LIN {X -0.046,Y -193.503,Z 910.176,A 0.000,B 0.000,C 90.000,E1 31.671} C_DIS
LIN {X 0.056,Y -188.124,Z 910.158,A 0.000,B 0.000,C 90.000,E1 28.359} C_DIS
LIN {X 0.087,Y -183.389,Z 910.139,A 0.000,B 0.000,C 90.000,E1 25.027} C_DIS
LIN {X -0.058,Y -179.252,Z 910.121,A 0.000,B 0.000,C 90.000,E1 21.716} C_DIS
LIN {X 0.005,Y -175.085,Z 910.097,A 0.000,B 0.000,C 90.000,E1 17.457} C_DIS
LIN {X 0.015,Y -172.098,Z 910.073,A 0.000,B 0.000,C 90.000,E1 13.175} C_DIS
LIN {X 0.060,Y -169.577,Z 910.040,A 0.000,B 0.000,C 90.000,E1 7.125} C_DIS
LIN {X 0.074,Y -170.579,Z 909.973,A 0.000,B 0.000,C 90.000,E1 355.179} C_DIS
LIN {X -0.024,Y -173.354,Z 909.945,A 0.000,B 0.000,C 90.000,E1 350.038} C_DIS
LIN {X -0.023,Y -176.708,Z 909.921,A 0.000,B 0.000,C 90.000,E1 345.755} C_DIS
LIN {X -0.051,Y -180.143,Z 909.902,A 0.000,B 0.000,C 90.000,E1 342.362} C_DIS
LIN {X 0.058,Y -184.300,Z 909.883,A 0.000,B 0.000,C 90.000,E1 338.954} C_DIS
LIN {X 0.061,Y -189.349,Z 909.865,A 0.000,B 0.000,C 90.000,E1 335.613} C_DIS
LIN {X -0.101,Y -195.206,Z 909.846,A 0.000,B 0.000,C 90.000,E1 332.359} C_DIS
LIN {X 0.047,Y -203.252,Z 909.824,A 0.000,B 0.000,C 90.000,E1 328.250} C_DIS
LIN {X 0.026,Y -210.215,Z 909.806,A 0.000,B 0.000,C 90.000,E1 325.055} C_DIS
LIN {X 0.020,Y -217.690,Z 909.788,A 0.000,B 0.000,C 90.000,E1 321.904} C_DIS
LIN {X 0.091,Y -226.821,Z 909.769,A 0.000,B 0.000,C 90.000,E1 318.405} C_DIS
LIN {X -0.057,Y -235.880,Z 909.752,A 0.000,B 0.000,C 90.000,E1 315.405} C_DIS
LIN {X 0.035,Y -245.907,Z 909.736,A 0.000,B 0.000,C 90.000,E1 312.405} C_DIS
LIN {X 0.057,Y -257.101,Z 909.719,A 0.000,B 0.000,C 90.000,E1 309.483} C_DIS
LIN {X -0.096,Y -269.400,Z 909.704,A 0.000,B 0.000,C 90.000,E1 306.664} C_DIS
LIN {X 0.083,Y -284.961,Z 909.686,A 0.000,B 0.000,C 90.000,E1 303.499} C_DIS
LIN {X 0.101,Y -301.959,Z 909.669,A 0.000,B 0.000,C 90.000,E1 300.463} C_DIS
LIN {X 0.029,Y -316.328,Z 909.657,A 0.000,B 0.000,C 90.000,E1 298.180} C_DIS
LIN {X -0.108,Y -329.854,Z 909.646,A 0.000,B 0.000,C 90.000,E1 296.283} C_DIS
LIN {X 0.009,Y -344.391,Z 909.635,A 0.000,B 0.000,C 90.000,E1 294.387} C_DIS
LIN {X 0.127,Y -367.738,Z 909.620,A 0.000,B 0.000,C 90.000,E1 291.663} C_DIS
LIN {X -0.013,Y -383.531,Z 909.611,A 0.000,B 0.000,C 90.000,E1 289.993} C_DIS
LIN {X -0.045,Y -401.556,Z 909.601,A 0.000,B 0.000,C 90.000,E1 288.109} C_DIS
LIN {X 0.162,Y -414.278,Z 909.593,A 0.000,B 0.000,C 90.000,E1 286.732} C_DIS
LIN {X 0.078,Y -424.276,Z 909.587,A 0.000,B 0.000,C 90.000,E1 285.662} C_DIS
LIN {X 0.006,Y -433.925,Z 909.581,A 0.000,B 0.000,C 90.000,E1 284.592} C_DIS
LIN {X 0.143,Y -445.299,Z 909.574,A 0.000,B 0.000,C 90.000,E1 283.244} C_DIS
LIN {X -0.231,Y -453.814,Z 909.568,A 0.000,B 0.000,C 90.000,E1 282.243} C_DIS
LIN {X -0.069,Y -461.769,Z 909.562,A 0.000,B 0.000,C 90.000,E1 281.186} C_DIS
LIN {X -0.046,Y -471.069,Z 909.555,A 0.000,B 0.000,C 90.000,E1 279.905} C_DIS
LIN {X -0.097,Y -476.327,Z 909.551,A 0.000,B 0.000,C 90.000,E1 279.151} C_DIS
LIN {X -0.096,Y -480.913,Z 909.547,A 0.000,B 0.000,C 90.000,E1 278.398} C_DIS
LIN {X -0.059,Y -484.725,Z 909.542,A 0.000,B 0.000,C 90.000,E1 277.644} C_DIS
LIN {X 0.126,Y -486.841,Z 909.540,A 0.000,B 0.000,C 90.000,E1 277.125} C_DIS
LIN {X -0.159,Y -488.603,Z 909.537,A 0.000,B 0.000,C 90.000,E1 276.663} C_DIS
LIN {X 0.047,Y -490.002,Z 909.534,A 0.000,B 0.000,C 90.000,E1 276.144} C_DIS
LIN {X -0.225,Y -491.072,Z 909.531,A 0.000,B 0.000,C 90.000,E1 275.682} C_DIS
LIN {X -0.002,Y -491.799,Z 909.529,A 0.000,B 0.000,C 90.000,E1 275.163} C_DIS
LIN {X 0.226,Y -492.165,Z 909.526,A 0.000,B 0.000,C 90.000,E1 274.645} C_DIS
LIN {X -0.070,Y -492.073,Z 909.523,A 0.000,B 0.000,C 90.000,E1 274.188} C_DIS
LIN {X 0.163,Y -491.518,Z 909.521,A 0.000,B 0.000,C 90.000,E1 273.669} C_DIS
LIN {X -0.127,Y -490.551,Z 909.518,A 0.000,B 0.000,C 90.000,E1 273.212} C_DIS
LIN {X 0.098,Y -489.016,Z 909.515,A 0.000,B 0.000,C 90.000,E1 272.694} C_DIS
LIN {X -0.195,Y -486.904,Z 909.512,A 0.000,B 0.000,C 90.000,E1 272.236} C_DIS
LIN {X 0.008,Y -484.104,Z 909.510,A 0.000,B 0.000,C 90.000,E1 271.718} C_DIS
LIN {X 0.173,Y -480.512,Z 909.507,A 0.000,B 0.000,C 90.000,E1 271.203} C_DIS
LIN {X -0.158,Y -476.050,Z 909.504,A 0.000,B 0.000,C 90.000,E1 270.745} C_DIS
LIN {X -0.032,Y -470.550,Z 909.501,A 0.000,B 0.000,C 90.000,E1 270.229} C_DIS
LIN {X -0.022,Y -464.477,Z 909.499,A 0.000,B 0.000,C 90.000,E1 269.771} C_DIS
LIN {X 0.008,Y -458.177,Z 909.497,A 0.000,B 0.000,C 90.000,E1 269.370} C_DIS
LIN {X -0.030,Y -451.593,Z 909.495,A 0.000,B 0.000,C 90.000,E1 269.026} C_DIS
LIN {X -0.148,Y -444.694,Z 909.493,A 0.000,B 0.000,C 90.000,E1 268.740} C_DIS
LIN {X 0.111,Y -437.786,Z 909.492,A 0.000,B 0.000,C 90.000,E1 268.453} C_DIS
LIN {X -0.214,Y -430.109,Z 909.490,A 0.000,B 0.000,C 90.000,E1 268.282} C_DIS
LIN {X -0.153,Y -421.664,Z 909.489,A 0.000,B 0.000,C 90.000,E1 268.108} C_DIS
LIN {X -0.161,Y -411.053,Z 909.489,A 0.000,B 0.000,C 90.000,E1 267.993} C_DIS
LIN {X 0.050,Y -404.242,Z 909.489,A 0.000,B 0.000,C 90.000,E1 267.936} C_DIS
LIN {X -0.007,Y -181.114,Z 909.489,A 0.000,B 0.000,C 90.000,E1 267.936} C_DIS
LIN {X 0.043,Y -180.906,Z 909.474,A 0.000,B 0.000,C 90.000,E1 265.355} C_DIS
LIN {X -0.063,Y -180.689,Z 909.470,A 0.000,B 0.000,C 90.000,E1 264.546} C_DIS
LIN {X 0.015,Y -178.773,Z 909.441,A 0.000,B 0.000,C 90.000,E1 259.454} C_DIS
LIN {X -0.082,Y -175.819,Z 909.413,A 0.000,B 0.000,C 90.000,E1 254.393} C_DIS
LIN {X 0.080,Y -172.006,Z 909.385,A 0.000,B 0.000,C 90.000,E1 249.209} C_DIS
LIN {X 0.055,Y -171.424,Z 909.380,A 0.000,B 0.000,C 90.000,E1 248.358} C_DIS
LIN {X -0.049,Y -167.662,Z 909.356,A 0.000,B 0.000,C 90.000,E1 244.076} C_DIS
LIN {X 0.039,Y -166.330,Z 909.346,A 0.000,B 0.000,C 90.000,E1 242.308} C_DIS
LIN {X 0.025,Y -163.069,Z 909.327,A 0.000,B 0.000,C 90.000,E1 238.820} C_DIS
LIN {X -0.064,Y -161.008,Z 909.312,A 0.000,B 0.000,C 90.000,E1 236.215} C_DIS
LIN {X 0.046,Y -157.752,Z 909.293,A 0.000,B 0.000,C 90.000,E1 232.637} C_DIS
LIN {X -0.016,Y -155.790,Z 909.278,A 0.000,B 0.000,C 90.000,E1 229.989} C_DIS
LIN {X 0.039,Y -152.044,Z 909.253,A 0.000,B 0.000,C 90.000,E1 225.486} C_DIS
LIN {X 0.057,Y -150.292,Z 909.238,A 0.000,B 0.000,C 90.000,E1 222.771} C_DIS
LIN {X -0.018,Y -147.040,Z 909.213,A 0.000,B 0.000,C 90.000,E1 218.257} C_DIS
LIN {X -0.025,Y -145.620,Z 909.197,A 0.000,B 0.000,C 90.000,E1 215.518} C_DIS
LIN {X -0.026,Y -143.004,Z 909.172,A 0.000,B 0.000,C 90.000,E1 210.924} C_DIS
LIN {X 0.031,Y -141.631,Z 909.151,A 0.000,B 0.000,C 90.000,E1 207.206} C_DIS
LIN {X -0.043,Y -139.435,Z 909.115,A 0.000,B 0.000,C 90.000,E1 200.737} C_DIS
LIN {X 0.011,Y -139.167,Z 909.105,A 0.000,B 0.000,C 90.000,E1 198.852} C_DIS
LIN {X 0.044,Y -138.316,Z 909.053,A 0.000,B 0.000,C 90.000,E1 189.500} C_DIS
LIN {X 0.055,Y -139.475,Z 909.006,A 0.000,B 0.000,C 90.000,E1 181.088} C_DIS
LIN {X -0.003,Y -141.056,Z 908.975,A 0.000,B 0.000,C 90.000,E1 175.527} C_DIS
LIN {X -0.050,Y -142.427,Z 908.960,A 0.000,B 0.000,C 90.000,E1 172.761} C_DIS
LIN {X 0.011,Y -144.665,Z 908.934,A 0.000,B 0.000,C 90.000,E1 168.117} C_DIS
LIN {X -0.005,Y -147.249,Z 908.914,A 0.000,B 0.000,C 90.000,E1 164.448} C_DIS
LIN {X 0.013,Y -150.566,Z 908.888,A 0.000,B 0.000,C 90.000,E1 159.880} C_DIS
LIN {X 0.092,Y -154.035,Z 908.868,A 0.000,B 0.000,C 90.000,E1 156.230} C_DIS
LIN {X 0.019,Y -157.451,Z 908.848,A 0.000,B 0.000,C 90.000,E1 152.666} C_DIS
LIN {X -0.032,Y -161.669,Z 908.828,A 0.000,B 0.000,C 90.000,E1 149.125} C_DIS
LIN {X -0.014,Y -165.864,Z 908.809,A 0.000,B 0.000,C 90.000,E1 145.595} C_DIS
LIN {X -0.023,Y -170.841,Z 908.789,A 0.000,B 0.000,C 90.000,E1 142.110} C_DIS
LIN {X 0.024,Y -175.711,Z 908.770,A 0.000,B 0.000,C 90.000,E1 138.647} C_DIS
LIN {X 0.015,Y -181.323,Z 908.751,A 0.000,B 0.000,C 90.000,E1 135.243} C_DIS
LIN {X -0.115,Y -186.807,Z 908.733,A 0.000,B 0.000,C 90.000,E1 131.919} C_DIS
LIN {X -0.043,Y -191.397,Z 908.719,A 0.000,B 0.000,C 90.000,E1 129.402} C_DIS
LIN {X -0.106,Y -193.630,Z 908.711,A 0.000,B 0.000,C 90.000,E1 128.096} C_DIS
LIN {X 0.018,Y -295.882,Z 908.711,A 0.000,B 0.000,C 90.000,E1 128.051} C_DIS
LIN {X 0.042,Y -297.426,Z 908.711,A 0.000,B 0.000,C 90.000,E1 128.016} C_DIS
LIN {X 0.058,Y -302.690,Z 908.710,A 0.000,B 0.000,C 90.000,E1 127.729} C_DIS
LIN {X 0.059,Y -305.900,Z 908.708,A 0.000,B 0.000,C 90.000,E1 127.397} C_DIS
LIN {X 0.025,Y -309.482,Z 908.705,A 0.000,B 0.000,C 90.000,E1 126.824} C_DIS
LIN {X -0.011,Y -310.894,Z 908.703,A 0.000,B 0.000,C 90.000,E1 126.503} C_DIS
LIN {X 0.040,Y -313.928,Z 908.697,A 0.000,B 0.000,C 90.000,E1 125.518} C_DIS
LIN {X -0.152,Y -324.459,Z 908.680,A 0.000,B 0.000,C 90.000,E1 122.339} C_DIS
LIN {X 0.085,Y -335.283,Z 908.664,A 0.000,B 0.000,C 90.000,E1 119.461} C_DIS
LIN {X -0.014,Y -347.491,Z 908.648,A 0.000,B 0.000,C 90.000,E1 116.693} C_DIS
LIN {X 0.092,Y -361.185,Z 908.633,A 0.000,B 0.000,C 90.000,E1 113.951} C_DIS
LIN {X 0.037,Y -374.708,Z 908.620,A 0.000,B 0.000,C 90.000,E1 111.589} C_DIS
LIN {X 0.048,Y -389.599,Z 908.607,A 0.000,B 0.000,C 90.000,E1 109.268} C_DIS
LIN {X -0.202,Y -405.967,Z 908.594,A 0.000,B 0.000,C 90.000,E1 107.040} C_DIS
LIN {X -0.180,Y -423.928,Z 908.582,A 0.000,B 0.000,C 90.000,E1 104.828} C_DIS
LIN {X 0.182,Y -443.471,Z 908.570,A 0.000,B 0.000,C 90.000,E1 102.647} C_DIS
LIN {X -0.136,Y -463.764,Z 908.559,A 0.000,B 0.000,C 90.000,E1 100.715} C_DIS
LIN {X -0.188,Y -468.605,Z 908.557,A 0.000,B 0.000,C 90.000,E1 100.254} C_DIS
LIN {X -0.152,Y -470.305,Z 908.556,A 0.000,B 0.000,C 90.000,E1 100.018} C_DIS
LIN {X 0.163,Y -471.726,Z 908.554,A 0.000,B 0.000,C 90.000,E1 99.726} C_DIS
LIN {X -0.066,Y -472.782,Z 908.553,A 0.000,B 0.000,C 90.000,E1 99.500} C_DIS
LIN {X 0.119,Y -474.016,Z 908.550,A 0.000,B 0.000,C 90.000,E1 98.973} C_DIS
LIN {X -0.235,Y -474.244,Z 908.547,A 0.000,B 0.000,C 90.000,E1 98.511} C_DIS
LIN {X -0.110,Y -473.506,Z 908.544,A 0.000,B 0.000,C 90.000,E1 97.992} C_DIS
LIN {X 0.079,Y -471.686,Z 908.542,A 0.000,B 0.000,C 90.000,E1 97.466} C_DIS
LIN {X -0.124,Y -470.263,Z 908.540,A 0.000,B 0.000,C 90.000,E1 97.239} C_DIS
LIN {X -0.226,Y -451.212,Z 908.523,A 0.000,B 0.000,C 90.000,E1 94.188} C_DIS
LIN {X 0.131,Y -441.906,Z 908.514,A 0.000,B 0.000,C 90.000,E1 92.579} C_DIS
LIN {X -0.144,Y -432.309,Z 908.506,A 0.000,B 0.000,C 90.000,E1 91.031} C_DIS
LIN {X -0.032,Y -421.046,Z 908.495,A 0.000,B 0.000,C 90.000,E1 89.141} C_DIS
LIN {X 0.025,Y -406.774,Z 908.482,A 0.000,B 0.000,C 90.000,E1 86.674} C_DIS
LIN {X 0.044,Y -395.625,Z 908.471,A 0.000,B 0.000,C 90.000,E1 84.723} C_DIS
LIN {X -0.101,Y -384.600,Z 908.460,A 0.000,B 0.000,C 90.000,E1 82.761} C_DIS
LIN {X -0.037,Y -373.487,Z 908.448,A 0.000,B 0.000,C 90.000,E1 80.735} C_DIS
LIN {X -0.156,Y -362.045,Z 908.437,A 0.000,B 0.000,C 90.000,E1 78.701} C_DIS
LIN {X 0.035,Y -352.171,Z 908.427,A 0.000,B 0.000,C 90.000,E1 76.881} C_DIS
LIN {X 0.034,Y -338.971,Z 908.414,A 0.000,B 0.000,C 90.000,E1 74.448} C_DIS
LIN {X 0.048,Y -323.458,Z 908.396,A 0.000,B 0.000,C 90.000,E1 71.329} C_DIS
LIN {X 0.141,Y -313.009,Z 908.384,A 0.000,B 0.000,C 90.000,E1 69.082} C_DIS
LIN {X -0.058,Y -302.709,Z 908.371,A 0.000,B 0.000,C 90.000,E1 66.847} C_DIS
LIN {X -0.075,Y -292.475,Z 908.358,A 0.000,B 0.000,C 90.000,E1 64.537} C_DIS
LIN {X 0.084,Y -283.578,Z 908.347,A 0.000,B 0.000,C 90.000,E1 62.487} C_DIS
LIN {X -0.098,Y -273.094,Z 908.334,A 0.000,B 0.000,C 90.000,E1 60.127} C_DIS
LIN {X -0.082,Y -261.439,Z 908.318,A 0.000,B 0.000,C 90.000,E1 57.327} C_DIS
LIN {X 0.076,Y -249.210,Z 908.300,A 0.000,B 0.000,C 90.000,E1 54.069} C_DIS
LIN {X -0.063,Y -238.537,Z 908.282,A 0.000,B 0.000,C 90.000,E1 50.803} C_DIS
LIN {X 0.123,Y -228.788,Z 908.263,A 0.000,B 0.000,C 90.000,E1 47.391} C_DIS
LIN {X 0.101,Y -220.820,Z 908.247,A 0.000,B 0.000,C 90.000,E1 44.352} C_DIS
LIN {X -0.100,Y -213.150,Z 908.229,A 0.000,B 0.000,C 90.000,E1 41.310} C_DIS
LIN {X -0.011,Y -206.212,Z 908.212,A 0.000,B 0.000,C 90.000,E1 38.141} C_DIS
LIN {X 0.004,Y -199.849,Z 908.194,A 0.000,B 0.000,C 90.000,E1 34.945} C_DIS
LIN {X -0.035,Y -193.833,Z 908.176,A 0.000,B 0.000,C 90.000,E1 31.720} C_DIS
LIN {X -0.022,Y -188.446,Z 908.158,A 0.000,B 0.000,C 90.000,E1 28.437} C_DIS
LIN {X 0.025,Y -183.686,Z 908.140,A 0.000,B 0.000,C 90.000,E1 25.103} C_DIS
LIN {X -0.040,Y -179.559,Z 908.121,A 0.000,B 0.000,C 90.000,E1 21.770} C_DIS
LIN {X 0.028,Y -175.398,Z 908.097,A 0.000,B 0.000,C 90.000,E1 17.511} C_DIS
LIN {X 0.003,Y -172.382,Z 908.074,A 0.000,B 0.000,C 90.000,E1 13.244} C_DIS
LIN {X -0.072,Y -169.842,Z 908.040,A 0.000,B 0.000,C 90.000,E1 7.239} C_DIS
LIN {X 0.067,Y -170.839,Z 907.973,A 0.000,B 0.000,C 90.000,E1 355.184} C_DIS
LIN {X -0.006,Y -173.615,Z 907.945,A 0.000,B 0.000,C 90.000,E1 350.038} C_DIS
LIN {X 0.002,Y -176.968,Z 907.921,A 0.000,B 0.000,C 90.000,E1 345.755} C_DIS
LIN {X -0.017,Y -180.400,Z 907.902,A 0.000,B 0.000,C 90.000,E1 342.362} C_DIS
LIN {X 0.098,Y -184.588,Z 907.883,A 0.000,B 0.000,C 90.000,E1 338.954} C_DIS
LIN {X -0.063,Y -189.647,Z 907.865,A 0.000,B 0.000,C 90.000,E1 335.665} C_DIS
LIN {X -0.043,Y -195.524,Z 907.846,A 0.000,B 0.000,C 90.000,E1 332.359} C_DIS
LIN {X 0.049,Y -201.909,Z 907.828,A 0.000,B 0.000,C 90.000,E1 329.076} C_DIS
LIN {X -0.006,Y -208.748,Z 907.810,A 0.000,B 0.000,C 90.000,E1 325.881} C_DIS
LIN {X -0.005,Y -216.054,Z 907.793,A 0.000,B 0.000,C 90.000,E1 322.718} C_DIS
LIN {X 0.008,Y -224.979,Z 907.773,A 0.000,B 0.000,C 90.000,E1 319.218} C_DIS
LIN {X -0.012,Y -233.794,Z 907.757,A 0.000,B 0.000,C 90.000,E1 316.176} C_DIS
LIN {X 0.022,Y -243.546,Z 907.740,A 0.000,B 0.000,C 90.000,E1 313.176} C_DIS
LIN {X -0.017,Y -254.456,Z 907.724,A 0.000,B 0.000,C 90.000,E1 310.253} C_DIS
LIN {X 0.089,Y -266.371,Z 907.708,A 0.000,B 0.000,C 90.000,E1 307.363} C_DIS
LIN {X -0.051,Y -281.476,Z 907.690,A 0.000,B 0.000,C 90.000,E1 304.246} C_DIS
LIN {X 0.007,Y -298.094,Z 907.673,A 0.000,B 0.000,C 90.000,E1 301.180} C_DIS
LIN {X -0.012,Y -311.998,Z 907.660,A 0.000,B 0.000,C 90.000,E1 298.871} C_DIS
LIN {X 0.053,Y -325.032,Z 907.650,A 0.000,B 0.000,C 90.000,E1 296.924} C_DIS
LIN {X 0.201,Y -344.108,Z 907.636,A 0.000,B 0.000,C 90.000,E1 294.387} C_DIS
LIN {X -0.048,Y -367.369,Z 907.621,A 0.000,B 0.000,C 90.000,E1 291.716} C_DIS
LIN {X 0.106,Y -383.190,Z 907.611,A 0.000,B 0.000,C 90.000,E1 289.993} C_DIS
LIN {X -0.124,Y -401.290,Z 907.601,A 0.000,B 0.000,C 90.000,E1 288.127} C_DIS
LIN {X 0.129,Y -413.978,Z 907.593,A 0.000,B 0.000,C 90.000,E1 286.749} C_DIS
LIN {X -0.027,Y -426.398,Z 907.586,A 0.000,B 0.000,C 90.000,E1 285.426} C_DIS
LIN {X -0.035,Y -435.890,Z 907.580,A 0.000,B 0.000,C 90.000,E1 284.356} C_DIS
LIN {X -0.087,Y -444.975,Z 907.574,A 0.000,B 0.000,C 90.000,E1 283.300} C_DIS
LIN {X -0.027,Y -453.529,Z 907.568,A 0.000,B 0.000,C 90.000,E1 282.243} C_DIS
LIN {X 0.135,Y -461.504,Z 907.562,A 0.000,B 0.000,C 90.000,E1 281.186} C_DIS
LIN {X 0.157,Y -470.835,Z 907.555,A 0.000,B 0.000,C 90.000,E1 279.905} C_DIS
LIN {X 0.106,Y -476.101,Z 907.551,A 0.000,B 0.000,C 90.000,E1 279.151} C_DIS
LIN {X 0.107,Y -480.746,Z 907.547,A 0.000,B 0.000,C 90.000,E1 278.398} C_DIS
LIN {X 0.145,Y -484.588,Z 907.543,A 0.000,B 0.000,C 90.000,E1 277.644} C_DIS
LIN {X -0.154,Y -486.729,Z 907.540,A 0.000,B 0.000,C 90.000,E1 277.182} C_DIS
LIN {X 0.045,Y -488.506,Z 907.537,A 0.000,B 0.000,C 90.000,E1 276.663} C_DIS
LIN {X -0.237,Y -489.968,Z 907.534,A 0.000,B 0.000,C 90.000,E1 276.201} C_DIS
LIN {X -0.022,Y -491.076,Z 907.532,A 0.000,B 0.000,C 90.000,E1 275.682} C_DIS
LIN {X 0.201,Y -491.804,Z 907.529,A 0.000,B 0.000,C 90.000,E1 275.163} C_DIS
LIN {X -0.060,Y -492.183,Z 907.526,A 0.000,B 0.000,C 90.000,E1 274.702} C_DIS
LIN {X 0.133,Y -492.129,Z 907.523,A 0.000,B 0.000,C 90.000,E1 274.188} C_DIS
LIN {X -0.125,Y -491.651,Z 907.521,A 0.000,B 0.000,C 90.000,E1 273.726} C_DIS
LIN {X 0.077,Y -490.690,Z 907.518,A 0.000,B 0.000,C 90.000,E1 273.212} C_DIS
LIN {X -0.186,Y -489.163,Z 907.515,A 0.000,B 0.000,C 90.000,E1 272.751} C_DIS
LIN {X 0.009,Y -487.145,Z 907.512,A 0.000,B 0.000,C 90.000,E1 272.236} C_DIS
LIN {X 0.211,Y -484.419,Z 907.510,A 0.000,B 0.000,C 90.000,E1 271.718} C_DIS
LIN {X -0.104,Y -480.930,Z 907.507,A 0.000,B 0.000,C 90.000,E1 271.260} C_DIS
LIN {X 0.046,Y -476.572,Z 907.504,A 0.000,B 0.000,C 90.000,E1 270.745} C_DIS
LIN {X 0.172,Y -471.201,Z 907.501,A 0.000,B 0.000,C 90.000,E1 270.229} C_DIS
LIN {X 0.151,Y -465.176,Z 907.499,A 0.000,B 0.000,C 90.000,E1 269.771} C_DIS
LIN {X 0.126,Y -458.928,Z 907.497,A 0.000,B 0.000,C 90.000,E1 269.370} C_DIS
LIN {X 0.063,Y -452.441,Z 907.495,A 0.000,B 0.000,C 90.000,E1 269.026} C_DIS
LIN {X -0.079,Y -445.631,Z 907.493,A 0.000,B 0.000,C 90.000,E1 268.740} C_DIS
LIN {X 0.129,Y -438.602,Z 907.492,A 0.000,B 0.000,C 90.000,E1 268.453} C_DIS
LIN {X -0.179,Y -431.227,Z 907.490,A 0.000,B 0.000,C 90.000,E1 268.282} C_DIS
LIN {X -0.137,Y -423.112,Z 907.489,A 0.000,B 0.000,C 90.000,E1 268.108} C_DIS
LIN {X -0.177,Y -413.915,Z 907.489,A 0.000,B 0.000,C 90.000,E1 267.993} C_DIS
LIN {X -0.073,Y -406.157,Z 907.488,A 0.000,B 0.000,C 90.000,E1 267.936} C_DIS
LIN {X -0.067,Y -181.111,Z 907.488,A 0.000,B 0.000,C 90.000,E1 267.936} C_DIS
LIN {X -0.001,Y -180.906,Z 907.474,A 0.000,B 0.000,C 90.000,E1 265.355} C_DIS
LIN {X 0.072,Y -180.681,Z 907.469,A 0.000,B 0.000,C 90.000,E1 264.489} C_DIS
LIN {X -0.029,Y -178.765,Z 907.441,A 0.000,B 0.000,C 90.000,E1 259.454} C_DIS
LIN {X 0.043,Y -175.811,Z 907.413,A 0.000,B 0.000,C 90.000,E1 254.338} C_DIS
LIN {X 0.037,Y -171.998,Z 907.385,A 0.000,B 0.000,C 90.000,E1 249.209} C_DIS
LIN {X 0.012,Y -171.411,Z 907.380,A 0.000,B 0.000,C 90.000,E1 248.358} C_DIS
LIN {X 0.060,Y -167.651,Z 907.356,A 0.000,B 0.000,C 90.000,E1 244.024} C_DIS
LIN {X 0.074,Y -166.315,Z 907.346,A 0.000,B 0.000,C 90.000,E1 242.281} C_DIS
LIN {X 0.068,Y -163.057,Z 907.327,A 0.000,B 0.000,C 90.000,E1 238.791} C_DIS
LIN {X 0.029,Y -160.993,Z 907.312,A 0.000,B 0.000,C 90.000,E1 236.167} C_DIS
LIN {X 0.006,Y -157.740,Z 907.292,A 0.000,B 0.000,C 90.000,E1 232.637} C_DIS
LIN {X -0.056,Y -155.778,Z 907.278,A 0.000,B 0.000,C 90.000,E1 229.989} C_DIS
LIN {X 0.000,Y -152.033,Z 907.253,A 0.000,B 0.000,C 90.000,E1 225.486} C_DIS
LIN {X 0.017,Y -150.281,Z 907.238,A 0.000,B 0.000,C 90.000,E1 222.771} C_DIS
LIN {X -0.056,Y -147.031,Z 907.212,A 0.000,B 0.000,C 90.000,E1 218.257} C_DIS
LIN {X -0.064,Y -145.612,Z 907.197,A 0.000,B 0.000,C 90.000,E1 215.518} C_DIS
LIN {X -0.064,Y -142.997,Z 907.172,A 0.000,B 0.000,C 90.000,E1 210.924} C_DIS
LIN {X -0.007,Y -141.624,Z 907.151,A 0.000,B 0.000,C 90.000,E1 207.206} C_DIS
LIN {X -0.081,Y -139.433,Z 907.115,A 0.000,B 0.000,C 90.000,E1 200.737} C_DIS
LIN {X -0.027,Y -139.163,Z 907.105,A 0.000,B 0.000,C 90.000,E1 198.852} C_DIS
LIN {X 0.011,Y -138.340,Z 907.058,A 0.000,B 0.000,C 90.000,E1 190.433} C_DIS
LIN {X 0.018,Y -139.478,Z 907.006,A 0.000,B 0.000,C 90.000,E1 181.088} C_DIS
LIN {X -0.042,Y -141.062,Z 906.975,A 0.000,B 0.000,C 90.000,E1 175.527} C_DIS
LIN {X 0.053,Y -142.435,Z 906.960,A 0.000,B 0.000,C 90.000,E1 172.704} C_DIS
LIN {X -0.027,Y -144.674,Z 906.934,A 0.000,B 0.000,C 90.000,E1 168.117} C_DIS
LIN {X -0.045,Y -147.261,Z 906.914,A 0.000,B 0.000,C 90.000,E1 164.448} C_DIS
LIN {X -0.027,Y -150.579,Z 906.888,A 0.000,B 0.000,C 90.000,E1 159.880} C_DIS
LIN {X 0.052,Y -154.050,Z 906.868,A 0.000,B 0.000,C 90.000,E1 156.230} C_DIS
LIN {X -0.021,Y -157.467,Z 906.848,A 0.000,B 0.000,C 90.000,E1 152.666} C_DIS
LIN {X 0.066,Y -161.689,Z 906.828,A 0.000,B 0.000,C 90.000,E1 149.076} C_DIS
LIN {X -0.057,Y -165.883,Z 906.809,A 0.000,B 0.000,C 90.000,E1 145.595} C_DIS
LIN {X -0.067,Y -170.863,Z 906.789,A 0.000,B 0.000,C 90.000,E1 142.110} C_DIS
LIN {X -0.020,Y -175.732,Z 906.770,A 0.000,B 0.000,C 90.000,E1 138.647} C_DIS
LIN {X -0.030,Y -181.343,Z 906.751,A 0.000,B 0.000,C 90.000,E1 135.243} C_DIS
LIN {X 0.104,Y -186.832,Z 906.733,A 0.000,B 0.000,C 90.000,E1 131.838} C_DIS
LIN {X 0.058,Y -191.420,Z 906.719,A 0.000,B 0.000,C 90.000,E1 129.358} C_DIS
LIN {X -0.031,Y -193.591,Z 906.712,A 0.000,B 0.000,C 90.000,E1 128.096} C_DIS
LIN {X -0.077,Y -294.987,Z 906.712,A 0.000,B 0.000,C 90.000,E1 128.096} C_DIS
LIN {X 0.005,Y -297.017,Z 906.711,A 0.000,B 0.000,C 90.000,E1 128.051} C_DIS
LIN {X -0.005,Y -300.818,Z 906.711,A 0.000,B 0.000,C 90.000,E1 127.890} C_DIS
LIN {X -0.015,Y -303.004,Z 906.710,A 0.000,B 0.000,C 90.000,E1 127.729} C_DIS
LIN {X 0.006,Y -306.889,Z 906.707,A 0.000,B 0.000,C 90.000,E1 127.282} C_DIS
LIN {X 0.114,Y -308.777,Z 906.705,A 0.000,B 0.000,C 90.000,E1 126.950} C_DIS
LIN {X -0.024,Y -310.260,Z 906.704,A 0.000,B 0.000,C 90.000,E1 126.664} C_DIS
LIN {X 0.198,Y -311.484,Z 906.702,A 0.000,B 0.000,C 90.000,E1 126.297} C_DIS
LIN {X -0.072,Y -322.769,Z 906.682,A 0.000,B 0.000,C 90.000,E1 122.801} C_DIS
LIN {X 0.114,Y -333.374,Z 906.666,A 0.000,B 0.000,C 90.000,E1 119.922} C_DIS
LIN {X 0.118,Y -345.345,Z 906.651,A 0.000,B 0.000,C 90.000,E1 117.129} C_DIS
LIN {X 0.162,Y -358.785,Z 906.636,A 0.000,B 0.000,C 90.000,E1 114.387} C_DIS
LIN {X 0.050,Y -372.062,Z 906.622,A 0.000,B 0.000,C 90.000,E1 112.025} C_DIS
LIN {X -0.003,Y -386.691,Z 906.609,A 0.000,B 0.000,C 90.000,E1 109.704} C_DIS
LIN {X -0.196,Y -402.774,Z 906.597,A 0.000,B 0.000,C 90.000,E1 107.457} C_DIS
LIN {X 0.152,Y -420.428,Z 906.584,A 0.000,B 0.000,C 90.000,E1 105.190} C_DIS
LIN {X -0.046,Y -439.725,Z 906.573,A 0.000,B 0.000,C 90.000,E1 103.063} C_DIS
LIN {X -0.171,Y -459.913,Z 906.561,A 0.000,B 0.000,C 90.000,E1 101.074} C_DIS
LIN {X -0.191,Y -467.568,Z 906.557,A 0.000,B 0.000,C 90.000,E1 100.366} C_DIS
LIN {X 0.173,Y -469.560,Z 906.556,A 0.000,B 0.000,C 90.000,E1 100.084} C_DIS
LIN {X 0.159,Y -471.076,Z 906.555,A 0.000,B 0.000,C 90.000,E1 99.849} C_DIS
LIN {X 0.013,Y -472.301,Z 906.553,A 0.000,B 0.000,C 90.000,E1 99.613} C_DIS
LIN {X -0.134,Y -473.198,Z 906.552,A 0.000,B 0.000,C 90.000,E1 99.378} C_DIS
LIN {X -0.024,Y -474.165,Z 906.549,A 0.000,B 0.000,C 90.000,E1 98.859} C_DIS
LIN {X 0.096,Y -474.150,Z 906.546,A 0.000,B 0.000,C 90.000,E1 98.341} C_DIS
LIN {X -0.181,Y -473.158,Z 906.544,A 0.000,B 0.000,C 90.000,E1 97.871} C_DIS
LIN {X -0.056,Y -471.019,Z 906.541,A 0.000,B 0.000,C 90.000,E1 97.352} C_DIS
LIN {X -0.137,Y -451.991,Z 906.524,A 0.000,B 0.000,C 90.000,E1 94.302} C_DIS
LIN {X -0.211,Y -442.727,Z 906.515,A 0.000,B 0.000,C 90.000,E1 92.751} C_DIS
LIN {X -0.033,Y -433.166,Z 906.506,A 0.000,B 0.000,C 90.000,E1 91.146} C_DIS
LIN {X 0.089,Y -421.884,Z 906.496,A 0.000,B 0.000,C 90.000,E1 89.255} C_DIS
LIN {X 0.170,Y -407.581,Z 906.482,A 0.000,B 0.000,C 90.000,E1 86.788} C_DIS
LIN {X -0.197,Y -396.422,Z 906.471,A 0.000,B 0.000,C 90.000,E1 84.894} C_DIS
LIN {X 0.072,Y -385.399,Z 906.460,A 0.000,B 0.000,C 90.000,E1 82.875} C_DIS
LIN {X 0.147,Y -374.296,Z 906.449,A 0.000,B 0.000,C 90.000,E1 80.849} C_DIS
LIN {X 0.048,Y -362.870,Z 906.438,A 0.000,B 0.000,C 90.000,E1 78.814} C_DIS
LIN {X -0.170,Y -353.042,Z 906.428,A 0.000,B 0.000,C 90.000,E1 77.061} C_DIS
LIN {X -0.146,Y -339.855,Z 906.414,A 0.000,B 0.000,C 90.000,E1 74.629} C_DIS
LIN {X 0.058,Y -322.758,Z 906.395,A 0.000,B 0.000,C 90.000,E1 71.167} C_DIS
LIN {X -0.056,Y -312.341,Z 906.383,A 0.000,B 0.000,C 90.000,E1 68.954} C_DIS
LIN {X 0.120,Y -303.528,Z 906.372,A 0.000,B 0.000,C 90.000,E1 66.975} C_DIS
LIN {X 0.105,Y -291.846,Z 906.358,A 0.000,B 0.000,C 90.000,E1 64.332} C_DIS
LIN {X -0.131,Y -282.955,Z 906.346,A 0.000,B 0.000,C 90.000,E1 62.359} C_DIS
LIN {X 0.053,Y -272.474,Z 906.333,A 0.000,B 0.000,C 90.000,E1 59.921} C_DIS
LIN {X -0.042,Y -259.467,Z 906.315,A 0.000,B 0.000,C 90.000,E1 56.786} C_DIS
LIN {X -0.015,Y -248.774,Z 906.299,A 0.000,B 0.000,C 90.000,E1 53.909} C_DIS
LIN {X 0.028,Y -238.171,Z 906.281,A 0.000,B 0.000,C 90.000,E1 50.598} C_DIS
LIN {X 0.033,Y -228.505,Z 906.262,A 0.000,B 0.000,C 90.000,E1 47.229} C_DIS
LIN {X 0.008,Y -220.587,Z 906.245,A 0.000,B 0.000,C 90.000,E1 44.190} C_DIS
LIN {X 0.105,Y -212.958,Z 906.228,A 0.000,B 0.000,C 90.000,E1 41.067} C_DIS
LIN {X 0.051,Y -206.088,Z 906.211,A 0.000,B 0.000,C 90.000,E1 37.935} C_DIS
LIN {X 0.063,Y -199.701,Z 906.193,A 0.000,B 0.000,C 90.000,E1 34.739} C_DIS
LIN {X -0.084,Y -193.741,Z 906.175,A 0.000,B 0.000,C 90.000,E1 31.544} C_DIS
LIN {X 0.026,Y -188.396,Z 906.157,A 0.000,B 0.000,C 90.000,E1 28.231} C_DIS
LIN {X 0.065,Y -183.651,Z 906.138,A 0.000,B 0.000,C 90.000,E1 24.899} C_DIS
LIN {X -0.075,Y -179.580,Z 906.120,A 0.000,B 0.000,C 90.000,E1 21.589} C_DIS
LIN {X -0.004,Y -175.483,Z 906.096,A 0.000,B 0.000,C 90.000,E1 17.330} C_DIS
LIN {X 0.027,Y -172.054,Z 906.068,A 0.000,B 0.000,C 90.000,E1 12.187} C_DIS
LIN {X 0.059,Y -169.750,Z 906.029,A 0.000,B 0.000,C 90.000,E1 5.277} C_DIS
LIN {X 0.075,Y -171.097,Z 905.973,A 0.000,B 0.000,C 90.000,E1 355.184} C_DIS
LIN {X 0.011,Y -173.878,Z 905.945,A 0.000,B 0.000,C 90.000,E1 350.038} C_DIS
LIN {X 0.028,Y -177.227,Z 905.921,A 0.000,B 0.000,C 90.000,E1 345.755} C_DIS
LIN {X 0.015,Y -180.664,Z 905.902,A 0.000,B 0.000,C 90.000,E1 342.362} C_DIS
LIN {X -0.100,Y -184.886,Z 905.883,A 0.000,B 0.000,C 90.000,E1 339.028} C_DIS
LIN {X -0.014,Y -189.967,Z 905.865,A 0.000,B 0.000,C 90.000,E1 335.665} C_DIS
LIN {X 0.015,Y -195.853,Z 905.846,A 0.000,B 0.000,C 90.000,E1 332.359} C_DIS
LIN {X -0.092,Y -203.915,Z 905.824,A 0.000,B 0.000,C 90.000,E1 328.329} C_DIS
LIN {X -0.029,Y -212.609,Z 905.802,A 0.000,B 0.000,C 90.000,E1 324.322} C_DIS
LIN {X -0.052,Y -221.198,Z 905.782,A 0.000,B 0.000,C 90.000,E1 320.803} C_DIS
LIN {X 0.007,Y -229.559,Z 905.765,A 0.000,B 0.000,C 90.000,E1 317.715} C_DIS
LIN {X 0.092,Y -238.809,Z 905.748,A 0.000,B 0.000,C 90.000,E1 314.676} C_DIS
LIN {X -0.085,Y -249.078,Z 905.732,A 0.000,B 0.000,C 90.000,E1 311.757} C_DIS
LIN {X 0.080,Y -261.953,Z 905.714,A 0.000,B 0.000,C 90.000,E1 308.463} C_DIS
LIN {X -0.025,Y -273.060,Z 905.700,A 0.000,B 0.000,C 90.000,E1 306.011} C_DIS
LIN {X 0.101,Y -288.779,Z 905.683,A 0.000,B 0.000,C 90.000,E1 302.880} C_DIS
LIN {X 0.074,Y -305.828,Z 905.666,A 0.000,B 0.000,C 90.000,E1 299.873} C_DIS
LIN {X 0.090,Y -320.444,Z 905.653,A 0.000,B 0.000,C 90.000,E1 297.590} C_DIS
LIN {X -0.047,Y -341.349,Z 905.638,A 0.000,B 0.000,C 90.000,E1 294.771} C_DIS
LIN {X 0.104,Y -367.032,Z 905.621,A 0.000,B 0.000,C 90.000,E1 291.716} C_DIS
LIN {X -0.032,Y -382.544,Z 905.611,A 0.000,B 0.000,C 90.000,E1 290.066} C_DIS
LIN {X 0.033,Y -400.849,Z 905.601,A 0.000,B 0.000,C 90.000,E1 288.127} C_DIS
LIN {X -0.039,Y -413.492,Z 905.593,A 0.000,B 0.000,C 90.000,E1 286.804} C_DIS
LIN {X 0.211,Y -425.946,Z 905.586,A 0.000,B 0.000,C 90.000,E1 285.426} C_DIS
LIN {X 0.153,Y -435.520,Z 905.580,A 0.000,B 0.000,C 90.000,E1 284.356} C_DIS
LIN {X 0.101,Y -444.657,Z 905.574,A 0.000,B 0.000,C 90.000,E1 283.300} C_DIS
LIN {X 0.160,Y -453.240,Z 905.568,A 0.000,B 0.000,C 90.000,E1 282.243} C_DIS
LIN {X -0.130,Y -461.239,Z 905.562,A 0.000,B 0.000,C 90.000,E1 281.243} C_DIS
LIN {X -0.119,Y -470.602,Z 905.555,A 0.000,B 0.000,C 90.000,E1 279.962} C_DIS
LIN {X -0.175,Y -475.882,Z 905.551,A 0.000,B 0.000,C 90.000,E1 279.208} C_DIS
LIN {X -0.179,Y -480.570,Z 905.547,A 0.000,B 0.000,C 90.000,E1 278.454} C_DIS
LIN {X -0.148,Y -484.438,Z 905.543,A 0.000,B 0.000,C 90.000,E1 277.701} C_DIS
LIN {X 0.035,Y -486.599,Z 905.540,A 0.000,B 0.000,C 90.000,E1 277.182} C_DIS
LIN {X -0.253,Y -488.407,Z 905.537,A 0.000,B 0.000,C 90.000,E1 276.720} C_DIS
LIN {X -0.048,Y -489.907,Z 905.534,A 0.000,B 0.000,C 90.000,E1 276.201} C_DIS
LIN {X 0.166,Y -491.011,Z 905.532,A 0.000,B 0.000,C 90.000,E1 275.682} C_DIS
LIN {X -0.100,Y -491.806,Z 905.529,A 0.000,B 0.000,C 90.000,E1 275.220} C_DIS
LIN {X 0.127,Y -492.224,Z 905.526,A 0.000,B 0.000,C 90.000,E1 274.702} C_DIS
LIN {X -0.170,Y -492.173,Z 905.523,A 0.000,B 0.000,C 90.000,E1 274.245} C_DIS
LIN {X 0.064,Y -491.741,Z 905.521,A 0.000,B 0.000,C 90.000,E1 273.726} C_DIS
LIN {X -0.225,Y -490.782,Z 905.518,A 0.000,B 0.000,C 90.000,E1 273.269} C_DIS
LIN {X 0.000,Y -489.340,Z 905.515,A 0.000,B 0.000,C 90.000,E1 272.751} C_DIS
LIN {X 0.196,Y -487.340,Z 905.513,A 0.000,B 0.000,C 90.000,E1 272.236} C_DIS
LIN {X -0.085,Y -484.727,Z 905.510,A 0.000,B 0.000,C 90.000,E1 271.776} C_DIS
LIN {X 0.083,Y -481.330,Z 905.507,A 0.000,B 0.000,C 90.000,E1 271.260} C_DIS
LIN {X 0.234,Y -477.053,Z 905.504,A 0.000,B 0.000,C 90.000,E1 270.745} C_DIS
LIN {X -0.111,Y -471.778,Z 905.502,A 0.000,B 0.000,C 90.000,E1 270.286} C_DIS
LIN {X -0.145,Y -465.900,Z 905.499,A 0.000,B 0.000,C 90.000,E1 269.828} C_DIS
LIN {X 0.218,Y -459.678,Z 905.497,A 0.000,B 0.000,C 90.000,E1 269.370} C_DIS
LIN {X 0.091,Y -453.097,Z 905.495,A 0.000,B 0.000,C 90.000,E1 269.026} C_DIS
LIN {X -0.092,Y -446.319,Z 905.493,A 0.000,B 0.000,C 90.000,E1 268.740} C_DIS
LIN {X 0.078,Y -439.191,Z 905.491,A 0.000,B 0.000,C 90.000,E1 268.453} C_DIS
LIN {X 0.165,Y -431.729,Z 905.490,A 0.000,B 0.000,C 90.000,E1 268.224} C_DIS
LIN {X 0.201,Y -423.694,Z 905.489,A 0.000,B 0.000,C 90.000,E1 268.051} C_DIS
LIN {X 0.147,Y -414.782,Z 905.489,A 0.000,B 0.000,C 90.000,E1 267.936} C_DIS
LIN {X 0.160,Y -405.067,Z 905.488,A 0.000,B 0.000,C 90.000,E1 267.879} C_DIS
LIN {X 0.037,Y -181.107,Z 905.488,A 0.000,B 0.000,C 90.000,E1 267.879} C_DIS
LIN {X -0.046,Y -180.906,Z 905.474,A 0.000,B 0.000,C 90.000,E1 265.355} C_DIS
LIN {X 0.027,Y -180.674,Z 905.469,A 0.000,B 0.000,C 90.000,E1 264.489} C_DIS
LIN {X -0.073,Y -178.756,Z 905.441,A 0.000,B 0.000,C 90.000,E1 259.454} C_DIS
LIN {X 0.000,Y -175.804,Z 905.413,A 0.000,B 0.000,C 90.000,E1 254.338} C_DIS
LIN {X -0.006,Y -171.989,Z 905.384,A 0.000,B 0.000,C 90.000,E1 249.209} C_DIS
LIN {X 0.031,Y -171.398,Z 905.380,A 0.000,B 0.000,C 90.000,E1 248.337} C_DIS
LIN {X 0.016,Y -167.640,Z 905.356,A 0.000,B 0.000,C 90.000,E1 244.024} C_DIS
LIN {X 0.031,Y -166.299,Z 905.346,A 0.000,B 0.000,C 90.000,E1 242.281} C_DIS
LIN {X 0.025,Y -163.045,Z 905.327,A 0.000,B 0.000,C 90.000,E1 238.791} C_DIS
LIN {X -0.013,Y -160.978,Z 905.312,A 0.000,B 0.000,C 90.000,E1 236.167} C_DIS
LIN {X -0.035,Y -157.727,Z 905.292,A 0.000,B 0.000,C 90.000,E1 232.637} C_DIS
LIN {X -0.097,Y -155.767,Z 905.278,A 0.000,B 0.000,C 90.000,E1 229.989} C_DIS
LIN {X -0.041,Y -152.022,Z 905.253,A 0.000,B 0.000,C 90.000,E1 225.486} C_DIS
LIN {X -0.023,Y -150.270,Z 905.238,A 0.000,B 0.000,C 90.000,E1 222.771} C_DIS
LIN {X -0.005,Y -147.022,Z 905.212,A 0.000,B 0.000,C 90.000,E1 218.222} C_DIS
LIN {X 0.016,Y -145.604,Z 905.197,A 0.000,B 0.000,C 90.000,E1 215.471} C_DIS
LIN {X 0.020,Y -142.990,Z 905.172,A 0.000,B 0.000,C 90.000,E1 210.875} C_DIS
LIN {X 0.020,Y -141.617,Z 905.151,A 0.000,B 0.000,C 90.000,E1 207.180} C_DIS
LIN {X 0.060,Y -139.430,Z 905.115,A 0.000,B 0.000,C 90.000,E1 200.663} C_DIS
LIN {X -0.020,Y -139.160,Z 905.105,A 0.000,B 0.000,C 90.000,E1 198.833} C_DIS
LIN {X -0.003,Y -138.342,Z 905.058,A 0.000,B 0.000,C 90.000,E1 190.423} C_DIS
LIN {X -0.021,Y -139.480,Z 905.006,A 0.000,B 0.000,C 90.000,E1 181.088} C_DIS
LIN {X 0.060,Y -141.069,Z 904.975,A 0.000,B 0.000,C 90.000,E1 175.469} C_DIS
LIN {X 0.015,Y -142.443,Z 904.959,A 0.000,B 0.000,C 90.000,E1 172.704} C_DIS
LIN {X -0.037,Y -144.683,Z 904.934,A 0.000,B 0.000,C 90.000,E1 168.105} C_DIS
LIN {X 0.058,Y -147.273,Z 904.913,A 0.000,B 0.000,C 90.000,E1 164.393} C_DIS
LIN {X -0.067,Y -150.592,Z 904.888,A 0.000,B 0.000,C 90.000,E1 159.880} C_DIS
LIN {X 0.011,Y -154.064,Z 904.868,A 0.000,B 0.000,C 90.000,E1 156.230} C_DIS
LIN {X 0.077,Y -157.483,Z 904.848,A 0.000,B 0.000,C 90.000,E1 152.615} C_DIS
LIN {X 0.024,Y -161.708,Z 904.828,A 0.000,B 0.000,C 90.000,E1 149.076} C_DIS
LIN {X 0.037,Y -165.902,Z 904.809,A 0.000,B 0.000,C 90.000,E1 145.548} C_DIS
LIN {X 0.025,Y -170.886,Z 904.789,A 0.000,B 0.000,C 90.000,E1 142.065} C_DIS
LIN {X 0.053,Y -175.755,Z 904.770,A 0.000,B 0.000,C 90.000,E1 138.609} C_DIS
LIN {X -0.075,Y -181.364,Z 904.751,A 0.000,B 0.000,C 90.000,E1 135.243} C_DIS
LIN {X 0.058,Y -186.858,Z 904.733,A 0.000,B 0.000,C 90.000,E1 131.838} C_DIS
LIN {X 0.012,Y -191.443,Z 904.719,A 0.000,B 0.000,C 90.000,E1 129.358} C_DIS
LIN {X 0.031,Y -193.560,Z 904.712,A 0.000,B 0.000,C 90.000,E1 128.096} C_DIS
LIN {X 0.012,Y -294.912,Z 904.712,A 0.000,B 0.000,C 90.000,E1 128.096} C_DIS
LIN {X -0.055,Y -296.170,Z 904.712,A 0.000,B 0.000,C 90.000,E1 128.096} C_DIS
LIN {X 0.047,Y -300.877,Z 904.711,A 0.000,B 0.000,C 90.000,E1 127.890} C_DIS
LIN {X -0.088,Y -303.290,Z 904.710,A 0.000,B 0.000,C 90.000,E1 127.729} C_DIS
LIN {X 0.099,Y -307.130,Z 904.707,A 0.000,B 0.000,C 90.000,E1 127.237} C_DIS
LIN {X -0.091,Y -308.999,Z 904.705,A 0.000,B 0.000,C 90.000,E1 126.950} C_DIS
LIN {X 0.152,Y -310.460,Z 904.703,A 0.000,B 0.000,C 90.000,E1 126.583} C_DIS
LIN {X -0.021,Y -312.589,Z 904.700,A 0.000,B 0.000,C 90.000,E1 125.964} C_DIS
LIN {X -0.064,Y -322.911,Z 904.682,A 0.000,B 0.000,C 90.000,E1 122.752} C_DIS
LIN {X 0.135,Y -333.536,Z 904.666,A 0.000,B 0.000,C 90.000,E1 119.873} C_DIS
LIN {X -0.154,Y -345.531,Z 904.651,A 0.000,B 0.000,C 90.000,E1 117.129} C_DIS
LIN {X -0.116,Y -358.995,Z 904.635,A 0.000,B 0.000,C 90.000,E1 114.387} C_DIS
LIN {X 0.112,Y -372.296,Z 904.622,A 0.000,B 0.000,C 90.000,E1 111.972} C_DIS
LIN {X 0.204,Y -386.950,Z 904.609,A 0.000,B 0.000,C 90.000,E1 109.631} C_DIS
LIN {X -0.105,Y -403.061,Z 904.597,A 0.000,B 0.000,C 90.000,E1 107.402} C_DIS
LIN {X -0.147,Y -420.746,Z 904.584,A 0.000,B 0.000,C 90.000,E1 105.190} C_DIS
LIN {X 0.084,Y -440.067,Z 904.572,A 0.000,B 0.000,C 90.000,E1 103.008} C_DIS
LIN {X 0.081,Y -460.265,Z 904.561,A 0.000,B 0.000,C 90.000,E1 101.007} C_DIS
LIN {X -0.015,Y -467.871,Z 904.557,A 0.000,B 0.000,C 90.000,E1 100.310} C_DIS
LIN {X -0.052,Y -469.809,Z 904.556,A 0.000,B 0.000,C 90.000,E1 100.074} C_DIS
LIN {X -0.172,Y -471.281,Z 904.555,A 0.000,B 0.000,C 90.000,E1 99.849} C_DIS
LIN {X 0.001,Y -473.306,Z 904.552,A 0.000,B 0.000,C 90.000,E1 99.321} C_DIS
LIN {X 0.107,Y -474.196,Z 904.549,A 0.000,B 0.000,C 90.000,E1 98.803} C_DIS
LIN {X -0.241,Y -474.110,Z 904.546,A 0.000,B 0.000,C 90.000,E1 98.341} C_DIS
LIN {X -0.048,Y -473.039,Z 904.543,A 0.000,B 0.000,C 90.000,E1 97.814} C_DIS
LIN {X -0.251,Y -472.087,Z 904.542,A 0.000,B 0.000,C 90.000,E1 97.587} C_DIS
LIN {X 0.076,Y -470.798,Z 904.541,A 0.000,B 0.000,C 90.000,E1 97.296} C_DIS
LIN {X 0.221,Y -450.234,Z 904.522,A 0.000,B 0.000,C 90.000,E1 93.955} C_DIS
LIN {X 0.082,Y -440.969,Z 904.513,A 0.000,B 0.000,C 90.000,E1 92.407} C_DIS
LIN {X -0.054,Y -429.761,Z 904.503,A 0.000,B 0.000,C 90.000,E1 90.573} C_DIS
LIN {X -0.002,Y -418.429,Z 904.493,A 0.000,B 0.000,C 90.000,E1 88.682} C_DIS
LIN {X -0.080,Y -405.756,Z 904.481,A 0.000,B 0.000,C 90.000,E1 86.502} C_DIS
LIN {X -0.045,Y -394.604,Z 904.470,A 0.000,B 0.000,C 90.000,E1 84.546} C_DIS
LIN {X 0.131,Y -383.531,Z 904.459,A 0.000,B 0.000,C 90.000,E1 82.534} C_DIS
LIN {X -0.159,Y -374.030,Z 904.449,A 0.000,B 0.000,C 90.000,E1 80.849} C_DIS
LIN {X 0.102,Y -362.632,Z 904.438,A 0.000,B 0.000,C 90.000,E1 78.757} C_DIS
LIN {X -0.044,Y -352.832,Z 904.428,A 0.000,B 0.000,C 90.000,E1 76.992} C_DIS
LIN {X -0.109,Y -339.692,Z 904.414,A 0.000,B 0.000,C 90.000,E1 74.574} C_DIS
LIN {X -0.120,Y -322.606,Z 904.395,A 0.000,B 0.000,C 90.000,E1 71.148} C_DIS
LIN {X -0.041,Y -312.202,Z 904.383,A 0.000,B 0.000,C 90.000,E1 68.901} C_DIS
LIN {X 0.127,Y -303.398,Z 904.372,A 0.000,B 0.000,C 90.000,E1 66.922} C_DIS
LIN {X 0.104,Y -291.721,Z 904.357,A 0.000,B 0.000,C 90.000,E1 64.280} C_DIS
LIN {X -0.006,Y -282.850,Z 904.346,A 0.000,B 0.000,C 90.000,E1 62.281} C_DIS
LIN {X 0.039,Y -272.388,Z 904.333,A 0.000,B 0.000,C 90.000,E1 59.871} C_DIS
LIN {X 0.077,Y -259.418,Z 904.315,A 0.000,B 0.000,C 90.000,E1 56.707} C_DIS
LIN {X -0.033,Y -247.537,Z 904.297,A 0.000,B 0.000,C 90.000,E1 53.497} C_DIS
LIN {X -0.058,Y -237.087,Z 904.279,A 0.000,B 0.000,C 90.000,E1 50.194} C_DIS
LIN {X -0.011,Y -228.576,Z 904.262,A 0.000,B 0.000,C 90.000,E1 47.187} C_DIS
LIN {X -0.036,Y -218.788,Z 904.241,A 0.000,B 0.000,C 90.000,E1 43.380} C_DIS
LIN {X 0.034,Y -211.302,Z 904.224,A 0.000,B 0.000,C 90.000,E1 40.253} C_DIS
LIN {X 0.103,Y -204.627,Z 904.206,A 0.000,B 0.000,C 90.000,E1 37.076} C_DIS
LIN {X -0.037,Y -198.286,Z 904.188,A 0.000,B 0.000,C 90.000,E1 33.913} C_DIS
LIN {X -0.049,Y -192.506,Z 904.170,A 0.000,B 0.000,C 90.000,E1 30.669} C_DIS
LIN {X -0.064,Y -187.327,Z 904.152,A 0.000,B 0.000,C 90.000,E1 27.385} C_DIS
LIN {X 0.037,Y -182.748,Z 904.134,A 0.000,B 0.000,C 90.000,E1 24.027} C_DIS
LIN {X 0.062,Y -177.983,Z 904.110,A 0.000,B 0.000,C 90.000,E1 19.812} C_DIS
LIN {X -0.079,Y -174.406,Z 904.087,A 0.000,B 0.000,C 90.000,E1 15.607} C_DIS
LIN {X 0.011,Y -171.468,Z 904.058,A 0.000,B 0.000,C 90.000,E1 10.433} C_DIS
LIN {X -0.081,Y -172.112,Z 903.964,A 0.000,B 0.000,C 90.000,E1 353.514} C_DIS
LIN {X -0.022,Y -175.370,Z 903.935,A 0.000,B 0.000,C 90.000,E1 348.342} C_DIS
LIN {X -0.093,Y -179.093,Z 903.911,A 0.000,B 0.000,C 90.000,E1 344.102} C_DIS
LIN {X 0.039,Y -182.959,Z 903.893,A 0.000,B 0.000,C 90.000,E1 340.678} C_DIS
LIN {X -0.065,Y -187.643,Z 903.874,A 0.000,B 0.000,C 90.000,E1 337.358} C_DIS
LIN {X -0.005,Y -193.175,Z 903.856,A 0.000,B 0.000,C 90.000,E1 334.024} C_DIS
LIN {X 0.111,Y -199.340,Z 903.838,A 0.000,B 0.000,C 90.000,E1 330.717} C_DIS
LIN {X -0.047,Y -205.907,Z 903.820,A 0.000,B 0.000,C 90.000,E1 327.533} C_DIS
LIN {X 0.056,Y -212.916,Z 903.802,A 0.000,B 0.000,C 90.000,E1 324.322} C_DIS
LIN {X 0.046,Y -221.459,Z 903.782,A 0.000,B 0.000,C 90.000,E1 320.803} C_DIS
LIN {X -0.113,Y -230.919,Z 903.763,A 0.000,B 0.000,C 90.000,E1 317.391} C_DIS
LIN {X 0.146,Y -241.509,Z 903.744,A 0.000,B 0.000,C 90.000,E1 313.947} C_DIS
LIN {X -0.132,Y -252.093,Z 903.728,A 0.000,B 0.000,C 90.000,E1 311.067} C_DIS
LIN {X -0.045,Y -265.219,Z 903.710,A 0.000,B 0.000,C 90.000,E1 307.810} C_DIS
LIN {X 0.072,Y -278.264,Z 903.694,A 0.000,B 0.000,C 90.000,E1 304.978} C_DIS
LIN {X -0.038,Y -294.320,Z 903.677,A 0.000,B 0.000,C 90.000,E1 301.926} C_DIS
LIN {X -0.072,Y -311.827,Z 903.661,A 0.000,B 0.000,C 90.000,E1 298.949} C_DIS
LIN {X 0.078,Y -326.998,Z 903.648,A 0.000,B 0.000,C 90.000,E1 296.668} C_DIS
LIN {X 0.133,Y -343.575,Z 903.636,A 0.000,B 0.000,C 90.000,E1 294.463} C_DIS
LIN {X -0.075,Y -366.677,Z 903.621,A 0.000,B 0.000,C 90.000,E1 291.770} C_DIS
LIN {X -0.088,Y -384.815,Z 903.610,A 0.000,B 0.000,C 90.000,E1 289.812} C_DIS
LIN {X 0.201,Y -402.836,Z 903.599,A 0.000,B 0.000,C 90.000,E1 287.873} C_DIS
LIN {X -0.007,Y -415.463,Z 903.592,A 0.000,B 0.000,C 90.000,E1 286.567} C_DIS
LIN {X 0.041,Y -425.489,Z 903.586,A 0.000,B 0.000,C 90.000,E1 285.481} C_DIS
LIN {X -0.027,Y -435.087,Z 903.580,A 0.000,B 0.000,C 90.000,E1 284.411} C_DIS
LIN {X -0.017,Y -444.182,Z 903.574,A 0.000,B 0.000,C 90.000,E1 283.355} C_DIS
LIN {X 0.033,Y -452.820,Z 903.568,A 0.000,B 0.000,C 90.000,E1 282.299} C_DIS
LIN {X 0.186,Y -460.883,Z 903.563,A 0.000,B 0.000,C 90.000,E1 281.243} C_DIS
LIN {X 0.198,Y -470.277,Z 903.555,A 0.000,B 0.000,C 90.000,E1 279.962} C_DIS
LIN {X 0.142,Y -475.592,Z 903.551,A 0.000,B 0.000,C 90.000,E1 279.208} C_DIS
LIN {X 0.139,Y -480.300,Z 903.547,A 0.000,B 0.000,C 90.000,E1 278.454} C_DIS
LIN {X 0.171,Y -484.201,Z 903.543,A 0.000,B 0.000,C 90.000,E1 277.701} C_DIS
LIN {X -0.130,Y -486.402,Z 903.540,A 0.000,B 0.000,C 90.000,E1 277.239} C_DIS
LIN {X 0.066,Y -488.274,Z 903.537,A 0.000,B 0.000,C 90.000,E1 276.720} C_DIS
LIN {X -0.217,Y -489.803,Z 903.535,A 0.000,B 0.000,C 90.000,E1 276.258} C_DIS
LIN {X -0.004,Y -490.984,Z 903.532,A 0.000,B 0.000,C 90.000,E1 275.739} C_DIS
LIN {X 0.218,Y -491.774,Z 903.529,A 0.000,B 0.000,C 90.000,E1 275.220} C_DIS
LIN {X -0.045,Y -492.226,Z 903.526,A 0.000,B 0.000,C 90.000,E1 274.759} C_DIS
LIN {X 0.148,Y -492.254,Z 903.524,A 0.000,B 0.000,C 90.000,E1 274.245} C_DIS
LIN {X -0.109,Y -491.848,Z 903.521,A 0.000,B 0.000,C 90.000,E1 273.784} C_DIS
LIN {X 0.093,Y -490.950,Z 903.518,A 0.000,B 0.000,C 90.000,E1 273.269} C_DIS
LIN {X -0.171,Y -489.557,Z 903.516,A 0.000,B 0.000,C 90.000,E1 272.808} C_DIS
LIN {X 0.027,Y -487.637,Z 903.513,A 0.000,B 0.000,C 90.000,E1 272.293} C_DIS
LIN {X 0.231,Y -485.104,Z 903.510,A 0.000,B 0.000,C 90.000,E1 271.776} C_DIS
LIN {X -0.082,Y -481.824,Z 903.507,A 0.000,B 0.000,C 90.000,E1 271.318} C_DIS
LIN {X 0.236,Y -479.908,Z 903.506,A 0.000,B 0.000,C 90.000,E1 271.031} C_DIS
LIN {X -0.098,Y -475.247,Z 903.503,A 0.000,B 0.000,C 90.000,E1 270.573} C_DIS
LIN {X 0.148,Y -469.788,Z 903.500,A 0.000,B 0.000,C 90.000,E1 270.057} C_DIS
LIN {X -0.203,Y -463.827,Z 903.498,A 0.000,B 0.000,C 90.000,E1 269.656} C_DIS
LIN {X -0.109,Y -457.497,Z 903.496,A 0.000,B 0.000,C 90.000,E1 269.255} C_DIS
LIN {X -0.078,Y -450.927,Z 903.494,A 0.000,B 0.000,C 90.000,E1 268.912} C_DIS
LIN {X -0.142,Y -444.007,Z 903.492,A 0.000,B 0.000,C 90.000,E1 268.625} C_DIS
LIN {X 0.162,Y -436.787,Z 903.491,A 0.000,B 0.000,C 90.000,E1 268.339} C_DIS
LIN {X -0.011,Y -429.300,Z 903.490,A 0.000,B 0.000,C 90.000,E1 268.165} C_DIS
LIN {X 0.146,Y -421.025,Z 903.489,A 0.000,B 0.000,C 90.000,E1 267.993} C_DIS
LIN {X 0.166,Y -410.535,Z 903.488,A 0.000,B 0.000,C 90.000,E1 267.879} C_DIS
LIN {X 0.041,Y -406.204,Z 903.488,A 0.000,B 0.000,C 90.000,E1 267.879} C_DIS
LIN {X 0.000,Y -181.105,Z 903.488,A 0.000,B 0.000,C 90.000,E1 267.879} C_DIS
LIN {X -0.086,Y -180.905,Z 903.474,A 0.000,B 0.000,C 90.000,E1 265.355} C_DIS
LIN {X -0.012,Y -180.667,Z 903.469,A 0.000,B 0.000,C 90.000,E1 264.489} C_DIS
LIN {X 0.062,Y -178.749,Z 903.441,A 0.000,B 0.000,C 90.000,E1 259.398} C_DIS
LIN {X -0.040,Y -175.796,Z 903.413,A 0.000,B 0.000,C 90.000,E1 254.338} C_DIS
LIN {X -0.045,Y -171.981,Z 903.384,A 0.000,B 0.000,C 90.000,E1 249.209} C_DIS
LIN {X -0.007,Y -171.386,Z 903.380,A 0.000,B 0.000,C 90.000,E1 248.337} C_DIS
LIN {X -0.022,Y -167.631,Z 903.356,A 0.000,B 0.000,C 90.000,E1 244.024} C_DIS
LIN {X -0.006,Y -166.286,Z 903.346,A 0.000,B 0.000,C 90.000,E1 242.281} C_DIS
LIN {X -0.013,Y -163.034,Z 903.327,A 0.000,B 0.000,C 90.000,E1 238.791} C_DIS
LIN {X 0.040,Y -160.964,Z 903.312,A 0.000,B 0.000,C 90.000,E1 236.135} C_DIS
LIN {X -0.073,Y -157.717,Z 903.292,A 0.000,B 0.000,C 90.000,E1 232.637} C_DIS
LIN {X 0.086,Y -155.756,Z 903.277,A 0.000,B 0.000,C 90.000,E1 229.908} C_DIS
LIN {X -0.077,Y -152.012,Z 903.253,A 0.000,B 0.000,C 90.000,E1 225.486} C_DIS
LIN {X -0.059,Y -150.259,Z 903.237,A 0.000,B 0.000,C 90.000,E1 222.771} C_DIS
LIN {X 0.075,Y -147.013,Z 903.212,A 0.000,B 0.000,C 90.000,E1 218.177} C_DIS
LIN {X -0.019,Y -145.597,Z 903.197,A 0.000,B 0.000,C 90.000,E1 215.471} C_DIS
LIN {X -0.015,Y -142.984,Z 903.172,A 0.000,B 0.000,C 90.000,E1 210.875} C_DIS
LIN {X -0.015,Y -141.611,Z 903.151,A 0.000,B 0.000,C 90.000,E1 207.180} C_DIS
LIN {X 0.026,Y -139.428,Z 903.115,A 0.000,B 0.000,C 90.000,E1 200.663} C_DIS
LIN {X 0.077,Y -139.156,Z 903.104,A 0.000,B 0.000,C 90.000,E1 198.779} C_DIS
LIN {X -0.037,Y -138.343,Z 903.058,A 0.000,B 0.000,C 90.000,E1 190.423} C_DIS
LIN {X -0.055,Y -139.482,Z 903.006,A 0.000,B 0.000,C 90.000,E1 181.088} C_DIS
LIN {X 0.026,Y -141.075,Z 902.975,A 0.000,B 0.000,C 90.000,E1 175.469} C_DIS
LIN {X -0.021,Y -142.450,Z 902.959,A 0.000,B 0.000,C 90.000,E1 172.704} C_DIS
LIN {X 0.070,Y -144.692,Z 902.934,A 0.000,B 0.000,C 90.000,E1 168.049} C_DIS
LIN {X 0.023,Y -147.284,Z 902.913,A 0.000,B 0.000,C 90.000,E1 164.393} C_DIS
LIN {X 0.038,Y -150.603,Z 902.888,A 0.000,B 0.000,C 90.000,E1 159.826} C_DIS
LIN {X -0.026,Y -154.077,Z 902.868,A 0.000,B 0.000,C 90.000,E1 156.230} C_DIS
LIN {X 0.040,Y -157.497,Z 902.848,A 0.000,B 0.000,C 90.000,E1 152.615} C_DIS
LIN {X -0.014,Y -161.725,Z 902.828,A 0.000,B 0.000,C 90.000,E1 149.076} C_DIS
LIN {X -0.001,Y -165.919,Z 902.809,A 0.000,B 0.000,C 90.000,E1 145.548} C_DIS
LIN {X -0.014,Y -170.906,Z 902.789,A 0.000,B 0.000,C 90.000,E1 142.065} C_DIS
LIN {X 0.012,Y -175.774,Z 902.770,A 0.000,B 0.000,C 90.000,E1 138.609} C_DIS
LIN {X 0.013,Y -181.383,Z 902.751,A 0.000,B 0.000,C 90.000,E1 135.202} C_DIS
LIN {X 0.017,Y -186.880,Z 902.732,A 0.000,B 0.000,C 90.000,E1 131.838} C_DIS
LIN {X -0.030,Y -191.463,Z 902.719,A 0.000,B 0.000,C 90.000,E1 129.358} C_DIS
LIN {X 0.080,Y -193.534,Z 902.712,A 0.000,B 0.000,C 90.000,E1 128.096} C_DIS
LIN {X 0.088,Y -295.184,Z 902.712,A 0.000,B 0.000,C 90.000,E1 128.096} C_DIS
LIN {X -0.118,Y -297.365,Z 902.712,A 0.000,B 0.000,C 90.000,E1 128.096} C_DIS
LIN {X -0.017,Y -301.244,Z 902.711,A 0.000,B 0.000,C 90.000,E1 127.890} C_DIS
LIN {X -0.154,Y -303.531,Z 902.709,A 0.000,B 0.000,C 90.000,E1 127.729} C_DIS
LIN {X -0.086,Y -307.390,Z 902.707,A 0.000,B 0.000,C 90.000,E1 127.237} C_DIS
LIN {X 0.120,Y -309.219,Z 902.705,A 0.000,B 0.000,C 90.000,E1 126.870} C_DIS
LIN {X -0.110,Y -310.645,Z 902.703,A 0.000,B 0.000,C 90.000,E1 126.583} C_DIS
LIN {X -0.099,Y -312.710,Z 902.700,A 0.000,B 0.000,C 90.000,E1 125.931} C_DIS
LIN {X 0.116,Y -323.054,Z 902.682,A 0.000,B 0.000,C 90.000,E1 122.673} C_DIS
LIN {X -0.136,Y -333.701,Z 902.666,A 0.000,B 0.000,C 90.000,E1 119.873} C_DIS
LIN {X 0.035,Y -345.719,Z 902.650,A 0.000,B 0.000,C 90.000,E1 117.052} C_DIS
LIN {X -0.071,Y -359.208,Z 902.635,A 0.000,B 0.000,C 90.000,E1 114.335} C_DIS
LIN {X -0.034,Y -372.534,Z 902.622,A 0.000,B 0.000,C 90.000,E1 111.950} C_DIS
LIN {X -0.088,Y -387.213,Z 902.609,A 0.000,B 0.000,C 90.000,E1 109.631} C_DIS
LIN {X 0.104,Y -403.352,Z 902.596,A 0.000,B 0.000,C 90.000,E1 107.330} C_DIS
LIN {X -0.043,Y -421.067,Z 902.584,A 0.000,B 0.000,C 90.000,E1 105.134} C_DIS
LIN {X -0.218,Y -440.413,Z 902.572,A 0.000,B 0.000,C 90.000,E1 103.008} C_DIS
LIN {X 0.244,Y -460.621,Z 902.561,A 0.000,B 0.000,C 90.000,E1 100.950} C_DIS
LIN {X 0.161,Y -468.165,Z 902.557,A 0.000,B 0.000,C 90.000,E1 100.254} C_DIS
LIN {X 0.094,Y -470.056,Z 902.556,A 0.000,B 0.000,C 90.000,E1 100.018} C_DIS
LIN {X -0.055,Y -471.490,Z 902.554,A 0.000,B 0.000,C 90.000,E1 99.792} C_DIS
LIN {X 0.121,Y -473.415,Z 902.552,A 0.000,B 0.000,C 90.000,E1 99.265} C_DIS
LIN {X -0.239,Y -474.228,Z 902.549,A 0.000,B 0.000,C 90.000,E1 98.803} C_DIS
LIN {X -0.050,Y -474.069,Z 902.546,A 0.000,B 0.000,C 90.000,E1 98.276} C_DIS
LIN {X 0.075,Y -472.918,Z 902.543,A 0.000,B 0.000,C 90.000,E1 97.757} C_DIS
LIN {X -0.128,Y -471.918,Z 902.542,A 0.000,B 0.000,C 90.000,E1 97.530} C_DIS
LIN {X 0.199,Y -470.572,Z 902.540,A 0.000,B 0.000,C 90.000,E1 97.239} C_DIS
LIN {X -0.116,Y -450.020,Z 902.522,A 0.000,B 0.000,C 90.000,E1 93.955} C_DIS
LIN {X 0.007,Y -442.342,Z 902.515,A 0.000,B 0.000,C 90.000,E1 92.636} C_DIS
LIN {X 0.176,Y -432.764,Z 902.506,A 0.000,B 0.000,C 90.000,E1 91.031} C_DIS
LIN {X 0.164,Y -423.103,Z 902.497,A 0.000,B 0.000,C 90.000,E1 89.427} C_DIS
LIN {X -0.161,Y -408.682,Z 902.483,A 0.000,B 0.000,C 90.000,E1 87.020} C_DIS
LIN {X -0.070,Y -397.555,Z 902.473,A 0.000,B 0.000,C 90.000,E1 85.065} C_DIS
LIN {X -0.167,Y -384.868,Z 902.460,A 0.000,B 0.000,C 90.000,E1 82.818} C_DIS
LIN {X -0.098,Y -373.758,Z 902.449,A 0.000,B 0.000,C 90.000,E1 80.792} C_DIS
LIN {X -0.185,Y -364.016,Z 902.439,A 0.000,B 0.000,C 90.000,E1 79.050} C_DIS
LIN {X 0.046,Y -354.247,Z 902.429,A 0.000,B 0.000,C 90.000,E1 77.229} C_DIS
LIN {X 0.099,Y -342.766,Z 902.417,A 0.000,B 0.000,C 90.000,E1 75.102} C_DIS
LIN {X 0.086,Y -325.454,Z 902.398,A 0.000,B 0.000,C 90.000,E1 71.692} C_DIS
LIN {X 0.042,Y -313.538,Z 902.384,A 0.000,B 0.000,C 90.000,E1 69.156} C_DIS
LIN {X -0.146,Y -303.258,Z 902.372,A 0.000,B 0.000,C 90.000,E1 66.922} C_DIS
LIN {X -0.033,Y -293.061,Z 902.359,A 0.000,B 0.000,C 90.000,E1 64.588} C_DIS
LIN {X 0.009,Y -284.236,Z 902.348,A 0.000,B 0.000,C 90.000,E1 62.564} C_DIS
LIN {X -0.156,Y -273.780,Z 902.334,A 0.000,B 0.000,C 90.000,E1 60.205} C_DIS
LIN {X -0.075,Y -260.785,Z 902.317,A 0.000,B 0.000,C 90.000,E1 57.041} C_DIS
LIN {X 0.068,Y -248.807,Z 902.299,A 0.000,B 0.000,C 90.000,E1 53.783} C_DIS
LIN {X -0.065,Y -239.370,Z 902.283,A 0.000,B 0.000,C 90.000,E1 50.884} C_DIS
LIN {X 0.031,Y -230.709,Z 902.266,A 0.000,B 0.000,C 90.000,E1 47.877} C_DIS
LIN {X 0.057,Y -222.734,Z 902.249,A 0.000,B 0.000,C 90.000,E1 44.838} C_DIS
LIN {X 0.050,Y -215.134,Z 902.232,A 0.000,B 0.000,C 90.000,E1 41.757} C_DIS
LIN {X 0.053,Y -208.049,Z 902.215,A 0.000,B 0.000,C 90.000,E1 38.624} C_DIS
LIN {X 0.075,Y -201.580,Z 902.197,A 0.000,B 0.000,C 90.000,E1 35.438} C_DIS
LIN {X 0.078,Y -195.483,Z 902.179,A 0.000,B 0.000,C 90.000,E1 32.212} C_DIS
LIN {X 0.061,Y -190.015,Z 902.161,A 0.000,B 0.000,C 90.000,E1 28.949} C_DIS
LIN {X -0.025,Y -185.127,Z 902.143,A 0.000,B 0.000,C 90.000,E1 25.668} C_DIS
LIN {X -0.053,Y -180.906,Z 902.124,A 0.000,B 0.000,C 90.000,E1 22.333} C_DIS
LIN {X -0.059,Y -177.363,Z 902.105,A 0.000,B 0.000,C 90.000,E1 18.960} C_DIS
LIN {X -0.098,Y -174.041,Z 902.082,A 0.000,B 0.000,C 90.000,E1 14.717} C_DIS
LIN {X -0.059,Y -171.368,Z 902.053,A 0.000,B 0.000,C 90.000,E1 9.557} C_DIS
LIN {X -0.069,Y -172.371,Z 901.964,A 0.000,B 0.000,C 90.000,E1 353.514} C_DIS
LIN {X -0.001,Y -175.633,Z 901.935,A 0.000,B 0.000,C 90.000,E1 348.342} C_DIS
LIN {X -0.063,Y -179.361,Z 901.912,A 0.000,B 0.000,C 90.000,E1 344.102} C_DIS
LIN {X -0.095,Y -183.252,Z 901.893,A 0.000,B 0.000,C 90.000,E1 340.732} C_DIS
LIN {X -0.019,Y -187.993,Z 901.874,A 0.000,B 0.000,C 90.000,E1 337.358} C_DIS
LIN {X 0.052,Y -193.513,Z 901.856,A 0.000,B 0.000,C 90.000,E1 334.024} C_DIS
LIN {X 0.027,Y -201.267,Z 901.833,A 0.000,B 0.000,C 90.000,E1 329.950} C_DIS
LIN {X -0.046,Y -207.903,Z 901.815,A 0.000,B 0.000,C 90.000,E1 326.755} C_DIS
LIN {X -0.012,Y -215.066,Z 901.798,A 0.000,B 0.000,C 90.000,E1 323.577} C_DIS
LIN {X 0.066,Y -222.753,Z 901.780,A 0.000,B 0.000,C 90.000,E1 320.436} C_DIS
LIN {X 0.106,Y -232.301,Z 901.761,A 0.000,B 0.000,C 90.000,E1 316.986} C_DIS
LIN {X 0.072,Y -243.016,Z 901.742,A 0.000,B 0.000,C 90.000,E1 313.623} C_DIS
LIN {X 0.017,Y -253.723,Z 901.726,A 0.000,B 0.000,C 90.000,E1 310.701} C_DIS
LIN {X 0.166,Y -266.961,Z 901.708,A 0.000,B 0.000,C 90.000,E1 307.443} C_DIS
LIN {X 0.049,Y -281.799,Z 901.691,A 0.000,B 0.000,C 90.000,E1 304.326} C_DIS
LIN {X 0.124,Y -298.065,Z 901.674,A 0.000,B 0.000,C 90.000,E1 301.258} C_DIS
LIN {X 0.161,Y -313.802,Z 901.659,A 0.000,B 0.000,C 90.000,E1 298.615} C_DIS
LIN {X -0.131,Y -331.402,Z 901.645,A 0.000,B 0.000,C 90.000,E1 296.104} C_DIS
LIN {X 0.020,Y -348.273,Z 901.633,A 0.000,B 0.000,C 90.000,E1 293.898} C_DIS
LIN {X -0.132,Y -368.727,Z 901.620,A 0.000,B 0.000,C 90.000,E1 291.535} C_DIS
LIN {X -0.028,Y -386.758,Z 901.609,A 0.000,B 0.000,C 90.000,E1 289.577} C_DIS
LIN {X -0.135,Y -402.405,Z 901.600,A 0.000,B 0.000,C 90.000,E1 287.946} C_DIS
LIN {X -0.239,Y -415.050,Z 901.592,A 0.000,B 0.000,C 90.000,E1 286.622} C_DIS
LIN {X 0.203,Y -425.128,Z 901.586,A 0.000,B 0.000,C 90.000,E1 285.481} C_DIS
LIN {X 0.026,Y -434.751,Z 901.580,A 0.000,B 0.000,C 90.000,E1 284.426} C_DIS
LIN {X 0.070,Y -443.981,Z 901.574,A 0.000,B 0.000,C 90.000,E1 283.355} C_DIS
LIN {X 0.119,Y -452.636,Z 901.568,A 0.000,B 0.000,C 90.000,E1 282.299} C_DIS
LIN {X -0.181,Y -460.725,Z 901.563,A 0.000,B 0.000,C 90.000,E1 281.299} C_DIS
LIN {X -0.180,Y -470.154,Z 901.556,A 0.000,B 0.000,C 90.000,E1 280.018} C_DIS
LIN {X 0.227,Y -475.475,Z 901.551,A 0.000,B 0.000,C 90.000,E1 279.208} C_DIS
LIN {X -0.121,Y -478.727,Z 901.549,A 0.000,B 0.000,C 90.000,E1 278.746} C_DIS
LIN {X -0.099,Y -482.899,Z 901.544,A 0.000,B 0.000,C 90.000,E1 277.992} C_DIS
LIN {X -0.045,Y -486.310,Z 901.540,A 0.000,B 0.000,C 90.000,E1 277.239} C_DIS
LIN {X 0.150,Y -488.224,Z 901.537,A 0.000,B 0.000,C 90.000,E1 276.720} C_DIS
LIN {X -0.133,Y -489.775,Z 901.535,A 0.000,B 0.000,C 90.000,E1 276.258} C_DIS
LIN {X 0.080,Y -490.980,Z 901.532,A 0.000,B 0.000,C 90.000,E1 275.739} C_DIS
LIN {X -0.188,Y -491.785,Z 901.529,A 0.000,B 0.000,C 90.000,E1 275.277} C_DIS
LIN {X 0.039,Y -492.223,Z 901.526,A 0.000,B 0.000,C 90.000,E1 274.759} C_DIS
LIN {X 0.232,Y -492.280,Z 901.524,A 0.000,B 0.000,C 90.000,E1 274.245} C_DIS
LIN {X -0.026,Y -491.918,Z 901.521,A 0.000,B 0.000,C 90.000,E1 273.784} C_DIS
LIN {X 0.175,Y -491.047,Z 901.518,A 0.000,B 0.000,C 90.000,E1 273.269} C_DIS
LIN {X -0.087,Y -489.690,Z 901.516,A 0.000,B 0.000,C 90.000,E1 272.808} C_DIS
LIN {X 0.110,Y -487.794,Z 901.513,A 0.000,B 0.000,C 90.000,E1 272.293} C_DIS
LIN {X -0.184,Y -485.295,Z 901.510,A 0.000,B 0.000,C 90.000,E1 271.835} C_DIS
LIN {X 0.158,Y -483.836,Z 901.509,A 0.000,B 0.000,C 90.000,E1 271.547} C_DIS
LIN {X -0.160,Y -480.218,Z 901.506,A 0.000,B 0.000,C 90.000,E1 271.088} C_DIS
LIN {X -0.013,Y -475.713,Z 901.503,A 0.000,B 0.000,C 90.000,E1 270.573} C_DIS
LIN {X 0.231,Y -470.310,Z 901.500,A 0.000,B 0.000,C 90.000,E1 270.057} C_DIS
LIN {X -0.137,Y -464.405,Z 901.498,A 0.000,B 0.000,C 90.000,E1 269.656} C_DIS
LIN {X -0.084,Y -458.114,Z 901.496,A 0.000,B 0.000,C 90.000,E1 269.255} C_DIS
LIN {X -0.099,Y -451.488,Z 901.494,A 0.000,B 0.000,C 90.000,E1 268.912} C_DIS
LIN {X -0.181,Y -444.614,Z 901.492,A 0.000,B 0.000,C 90.000,E1 268.625} C_DIS
LIN {X 0.118,Y -437.383,Z 901.491,A 0.000,B 0.000,C 90.000,E1 268.339} C_DIS
LIN {X -0.068,Y -429.967,Z 901.490,A 0.000,B 0.000,C 90.000,E1 268.165} C_DIS
LIN {X 0.066,Y -421.788,Z 901.489,A 0.000,B 0.000,C 90.000,E1 267.993} C_DIS
LIN {X 0.085,Y -412.088,Z 901.488,A 0.000,B 0.000,C 90.000,E1 267.879} C_DIS
LIN {X -0.101,Y -406.903,Z 901.488,A 0.000,B 0.000,C 90.000,E1 267.879} C_DIS
LIN {X -0.065,Y -181.101,Z 901.488,A 0.000,B 0.000,C 90.000,E1 267.879} C_DIS
LIN {X 0.073,Y -180.855,Z 901.472,A 0.000,B 0.000,C 90.000,E1 264.951} C_DIS
LIN {X -0.053,Y -178.968,Z 901.444,A 0.000,B 0.000,C 90.000,E1 259.926} C_DIS
LIN {X -0.042,Y -177.921,Z 901.435,A 0.000,B 0.000,C 90.000,E1 258.229} C_DIS
LIN {X -0.027,Y -175.558,Z 901.411,A 0.000,B 0.000,C 90.000,E1 253.976} C_DIS
LIN {X -0.020,Y -172.288,Z 901.387,A 0.000,B 0.000,C 90.000,E1 249.699} C_DIS
LIN {X -0.042,Y -171.766,Z 901.382,A 0.000,B 0.000,C 90.000,E1 248.847} C_DIS
LIN {X 0.037,Y -167.367,Z 901.354,A 0.000,B 0.000,C 90.000,E1 243.640} C_DIS
LIN {X -0.031,Y -166.757,Z 901.349,A 0.000,B 0.000,C 90.000,E1 242.794} C_DIS
LIN {X 0.029,Y -162.737,Z 901.325,A 0.000,B 0.000,C 90.000,E1 238.408} C_DIS
LIN {X 0.090,Y -161.427,Z 901.315,A 0.000,B 0.000,C 90.000,E1 236.628} C_DIS
LIN {X -0.089,Y -157.420,Z 901.290,A 0.000,B 0.000,C 90.000,E1 232.271} C_DIS
LIN {X 0.063,Y -155.424,Z 901.275,A 0.000,B 0.000,C 90.000,E1 229.542} C_DIS
LIN {X -0.006,Y -151.749,Z 901.250,A 0.000,B 0.000,C 90.000,E1 225.081} C_DIS
LIN {X 0.005,Y -149.948,Z 901.235,A 0.000,B 0.000,C 90.000,E1 222.366} C_DIS
LIN {X 0.033,Y -146.792,Z 901.210,A 0.000,B 0.000,C 90.000,E1 217.810} C_DIS
LIN {X -0.066,Y -145.367,Z 901.195,A 0.000,B 0.000,C 90.000,E1 215.105} C_DIS
LIN {X 0.051,Y -142.432,Z 901.164,A 0.000,B 0.000,C 90.000,E1 209.539} C_DIS
LIN {X -0.026,Y -141.422,Z 901.149,A 0.000,B 0.000,C 90.000,E1 206.796} C_DIS
LIN {X -0.044,Y -139.363,Z 901.113,A 0.000,B 0.000,C 90.000,E1 200.301} C_DIS
LIN {X 0.074,Y -138.806,Z 901.097,A 0.000,B 0.000,C 90.000,E1 197.457} C_DIS
LIN {X -0.008,Y -138.350,Z 901.056,A 0.000,B 0.000,C 90.000,E1 190.018} C_DIS
LIN {X -0.032,Y -139.544,Z 901.004,A 0.000,B 0.000,C 90.000,E1 180.688} C_DIS
LIN {X 0.061,Y -141.244,Z 900.973,A 0.000,B 0.000,C 90.000,E1 175.065} C_DIS
LIN {X 0.020,Y -142.613,Z 900.957,A 0.000,B 0.000,C 90.000,E1 172.299} C_DIS
LIN {X -0.028,Y -144.929,Z 900.932,A 0.000,B 0.000,C 90.000,E1 167.701} C_DIS
LIN {X -0.036,Y -147.558,Z 900.911,A 0.000,B 0.000,C 90.000,E1 164.031} C_DIS
LIN {X -0.004,Y -150.163,Z 900.891,A 0.000,B 0.000,C 90.000,E1 160.369} C_DIS
LIN {X 0.005,Y -153.536,Z 900.871,A 0.000,B 0.000,C 90.000,E1 156.741} C_DIS
LIN {X 0.057,Y -156.954,Z 900.851,A 0.000,B 0.000,C 90.000,E1 153.127} C_DIS
LIN {X -0.007,Y -161.060,Z 900.831,A 0.000,B 0.000,C 90.000,E1 149.587} C_DIS
LIN {X 0.078,Y -163.168,Z 900.821,A 0.000,B 0.000,C 90.000,E1 147.788} C_DIS
LIN {X -0.052,Y -167.587,Z 900.802,A 0.000,B 0.000,C 90.000,E1 144.322} C_DIS
LIN {X -0.006,Y -171.416,Z 900.787,A 0.000,B 0.000,C 90.000,E1 141.698} C_DIS
LIN {X 0.033,Y -176.333,Z 900.768,A 0.000,B 0.000,C 90.000,E1 138.243} C_DIS
LIN {X -0.099,Y -180.623,Z 900.754,A 0.000,B 0.000,C 90.000,E1 135.729} C_DIS
LIN {X 0.015,Y -186.024,Z 900.735,A 0.000,B 0.000,C 90.000,E1 132.324} C_DIS
LIN {X -0.068,Y -190.660,Z 900.721,A 0.000,B 0.000,C 90.000,E1 129.850} C_DIS
LIN {X -0.006,Y -193.499,Z 900.712,A 0.000,B 0.000,C 90.000,E1 128.141} C_DIS
LIN {X 0.170,Y -295.173,Z 900.712,A 0.000,B 0.000,C 90.000,E1 128.096} C_DIS
LIN {X 0.063,Y -296.560,Z 900.712,A 0.000,B 0.000,C 90.000,E1 128.096} C_DIS
LIN {X -0.080,Y -300.925,Z 900.711,A 0.000,B 0.000,C 90.000,E1 127.935} C_DIS
LIN {X 0.014,Y -303.303,Z 900.710,A 0.000,B 0.000,C 90.000,E1 127.729} C_DIS
LIN {X -0.038,Y -306.534,Z 900.708,A 0.000,B 0.000,C 90.000,E1 127.363} C_DIS
LIN {X 0.045,Y -308.482,Z 900.706,A 0.000,B 0.000,C 90.000,E1 127.030} C_DIS
LIN {X 0.067,Y -310.002,Z 900.704,A 0.000,B 0.000,C 90.000,E1 126.710} C_DIS
LIN {X 0.103,Y -311.236,Z 900.702,A 0.000,B 0.000,C 90.000,E1 126.377} C_DIS
LIN {X 0.090,Y -322.500,Z 900.682,A 0.000,B 0.000,C 90.000,E1 122.832} C_DIS
LIN {X -0.002,Y -333.076,Z 900.667,A 0.000,B 0.000,C 90.000,E1 120.001} C_DIS
LIN {X -0.003,Y -345.017,Z 900.651,A 0.000,B 0.000,C 90.000,E1 117.206} C_DIS
LIN {X 0.034,Y -358.424,Z 900.636,A 0.000,B 0.000,C 90.000,E1 114.463} C_DIS
LIN {X 0.056,Y -371.671,Z 900.623,A 0.000,B 0.000,C 90.000,E1 112.078} C_DIS
LIN {X -0.013,Y -386.266,Z 900.610,A 0.000,B 0.000,C 90.000,E1 109.758} C_DIS
LIN {X 0.162,Y -402.314,Z 900.597,A 0.000,B 0.000,C 90.000,E1 107.457} C_DIS
LIN {X 0.109,Y -419.931,Z 900.585,A 0.000,B 0.000,C 90.000,E1 105.245} C_DIS
LIN {X -0.116,Y -439.197,Z 900.573,A 0.000,B 0.000,C 90.000,E1 103.119} C_DIS
LIN {X 0.170,Y -459.372,Z 900.562,A 0.000,B 0.000,C 90.000,E1 101.074} C_DIS
LIN {X 0.143,Y -467.077,Z 900.558,A 0.000,B 0.000,C 90.000,E1 100.366} C_DIS
LIN {X 0.068,Y -469.176,Z 900.556,A 0.000,B 0.000,C 90.000,E1 100.141} C_DIS
LIN {X 0.077,Y -470.769,Z 900.555,A 0.000,B 0.000,C 90.000,E1 99.905} C_DIS
LIN {X -0.070,Y -472.075,Z 900.554,A 0.000,B 0.000,C 90.000,E1 99.670} C_DIS
LIN {X 0.247,Y -473.040,Z 900.552,A 0.000,B 0.000,C 90.000,E1 99.378} C_DIS
LIN {X -0.111,Y -474.121,Z 900.549,A 0.000,B 0.000,C 90.000,E1 98.916} C_DIS
LIN {X 0.007,Y -474.211,Z 900.547,A 0.000,B 0.000,C 90.000,E1 98.398} C_DIS
LIN {X 0.198,Y -473.330,Z 900.544,A 0.000,B 0.000,C 90.000,E1 97.871} C_DIS
LIN {X -0.146,Y -471.333,Z 900.541,A 0.000,B 0.000,C 90.000,E1 97.409} C_DIS
LIN {X 0.213,Y -458.507,Z 900.530,A 0.000,B 0.000,C 90.000,E1 95.334} C_DIS
LIN {X -0.031,Y -444.743,Z 900.517,A 0.000,B 0.000,C 90.000,E1 93.037} C_DIS
LIN {X 0.177,Y -435.258,Z 900.508,A 0.000,B 0.000,C 90.000,E1 91.432} C_DIS
LIN {X 0.207,Y -425.619,Z 900.499,A 0.000,B 0.000,C 90.000,E1 89.828} C_DIS
LIN {X 0.033,Y -409.521,Z 900.484,A 0.000,B 0.000,C 90.000,E1 87.135} C_DIS
LIN {X 0.058,Y -399.964,Z 900.475,A 0.000,B 0.000,C 90.000,E1 85.469} C_DIS
LIN {X 0.009,Y -387.273,Z 900.462,A 0.000,B 0.000,C 90.000,E1 83.223} C_DIS
LIN {X 0.127,Y -376.175,Z 900.451,A 0.000,B 0.000,C 90.000,E1 81.197} C_DIS
LIN {X 0.081,Y -366.523,Z 900.441,A 0.000,B 0.000,C 90.000,E1 79.454} C_DIS
LIN {X -0.115,Y -355.140,Z 900.430,A 0.000,B 0.000,C 90.000,E1 77.409} C_DIS
LIN {X -0.041,Y -343.690,Z 900.418,A 0.000,B 0.000,C 90.000,E1 75.283} C_DIS
LIN {X -0.019,Y -326.323,Z 900.399,A 0.000,B 0.000,C 90.000,E1 71.873} C_DIS
LIN {X -0.038,Y -314.418,Z 900.385,A 0.000,B 0.000,C 90.000,E1 69.337} C_DIS
LIN {X 0.076,Y -304.110,Z 900.373,A 0.000,B 0.000,C 90.000,E1 67.050} C_DIS
LIN {X 0.072,Y -292.476,Z 900.358,A 0.000,B 0.000,C 90.000,E1 64.409} C_DIS
LIN {X -0.025,Y -283.649,Z 900.347,A 0.000,B 0.000,C 90.000,E1 62.410} C_DIS
LIN {X 0.040,Y -273.212,Z 900.333,A 0.000,B 0.000,C 90.000,E1 59.999} C_DIS
LIN {X 0.104,Y -260.294,Z 900.316,A 0.000,B 0.000,C 90.000,E1 56.834} C_DIS
LIN {X 0.020,Y -248.425,Z 900.298,A 0.000,B 0.000,C 90.000,E1 53.623} C_DIS
LIN {X -0.128,Y -237.945,Z 900.280,A 0.000,B 0.000,C 90.000,E1 50.356} C_DIS
LIN {X 0.096,Y -229.458,Z 900.263,A 0.000,B 0.000,C 90.000,E1 47.310} C_DIS
LIN {X 0.093,Y -221.607,Z 900.246,A 0.000,B 0.000,C 90.000,E1 44.271} C_DIS
LIN {X -0.089,Y -214.080,Z 900.229,A 0.000,B 0.000,C 90.000,E1 41.229} C_DIS
LIN {X -0.107,Y -207.130,Z 900.211,A 0.000,B 0.000,C 90.000,E1 38.096} C_DIS
LIN {X -0.062,Y -200.706,Z 900.194,A 0.000,B 0.000,C 90.000,E1 34.898} C_DIS
LIN {X -0.072,Y -194.709,Z 900.176,A 0.000,B 0.000,C 90.000,E1 31.671} C_DIS
LIN {X 0.060,Y -189.343,Z 900.158,A 0.000,B 0.000,C 90.000,E1 28.359} C_DIS
LIN {X -0.046,Y -184.556,Z 900.139,A 0.000,B 0.000,C 90.000,E1 25.079} C_DIS
LIN {X 0.033,Y -179.543,Z 900.116,A 0.000,B 0.000,C 90.000,E1 20.865} C_DIS
LIN {X 0.052,Y -175.659,Z 900.092,A 0.000,B 0.000,C 90.000,E1 16.622} C_DIS
LIN {X -0.076,Y -172.478,Z 900.064,A 0.000,B 0.000,C 90.000,E1 11.535} C_DIS
LIN {X -0.082,Y -170.423,Z 900.021,A 0.000,B 0.000,C 90.000,E1 3.784} C_DIS
LIN {X -0.072,Y -171.900,Z 899.973,A 0.000,B 0.000,C 90.000,E1 355.241} C_DIS
LIN {X 0.065,Y -174.660,Z 899.945,A 0.000,B 0.000,C 90.000,E1 350.038} C_DIS
LIN {X -0.064,Y -178.032,Z 899.921,A 0.000,B 0.000,C 90.000,E1 345.811} C_DIS
LIN {X -0.057,Y -181.529,Z 899.902,A 0.000,B 0.000,C 90.000,E1 342.417} C_DIS
LIN {X 0.026,Y -185.842,Z 899.884,A 0.000,B 0.000,C 90.000,E1 339.028} C_DIS
LIN {X -0.035,Y -191.004,Z 899.865,A 0.000,B 0.000,C 90.000,E1 335.717} C_DIS
LIN {X 0.026,Y -196.900,Z 899.847,A 0.000,B 0.000,C 90.000,E1 332.410} C_DIS
LIN {X -0.042,Y -204.836,Z 899.824,A 0.000,B 0.000,C 90.000,E1 328.377} C_DIS
LIN {X -0.022,Y -211.734,Z 899.807,A 0.000,B 0.000,C 90.000,E1 325.182} C_DIS
LIN {X 0.014,Y -219.117,Z 899.789,A 0.000,B 0.000,C 90.000,E1 322.029} C_DIS
LIN {X -0.018,Y -228.191,Z 899.770,A 0.000,B 0.000,C 90.000,E1 318.566} C_DIS
LIN {X -0.136,Y -237.192,Z 899.753,A 0.000,B 0.000,C 90.000,E1 315.567} C_DIS
LIN {X 0.153,Y -247.116,Z 899.736,A 0.000,B 0.000,C 90.000,E1 312.528} C_DIS
LIN {X 0.072,Y -259.657,Z 899.718,A 0.000,B 0.000,C 90.000,E1 309.277} C_DIS
LIN {X -0.011,Y -271.903,Z 899.703,A 0.000,B 0.000,C 90.000,E1 306.457} C_DIS
LIN {X -0.146,Y -287.119,Z 899.685,A 0.000,B 0.000,C 90.000,E1 303.372} C_DIS
LIN {X -0.084,Y -303.760,Z 899.668,A 0.000,B 0.000,C 90.000,E1 300.335} C_DIS
LIN {X -0.028,Y -315.805,Z 899.658,A 0.000,B 0.000,C 90.000,E1 298.359} C_DIS
LIN {X 0.021,Y -333.473,Z 899.643,A 0.000,B 0.000,C 90.000,E1 295.796} C_DIS
LIN {X 0.002,Y -358.147,Z 899.626,A 0.000,B 0.000,C 90.000,E1 292.717} C_DIS
LIN {X -0.082,Y -378.681,Z 899.613,A 0.000,B 0.000,C 90.000,E1 290.429} C_DIS
LIN {X -0.129,Y -394.250,Z 899.604,A 0.000,B 0.000,C 90.000,E1 288.779} C_DIS
LIN {X 0.028,Y -407.139,Z 899.597,A 0.000,B 0.000,C 90.000,E1 287.402} C_DIS
LIN {X -0.172,Y -419.875,Z 899.589,A 0.000,B 0.000,C 90.000,E1 286.079} C_DIS
LIN {X 0.164,Y -429.766,Z 899.583,A 0.000,B 0.000,C 90.000,E1 284.954} C_DIS
LIN {X 0.152,Y -439.255,Z 899.577,A 0.000,B 0.000,C 90.000,E1 283.883} C_DIS
LIN {X 0.144,Y -448.195,Z 899.571,A 0.000,B 0.000,C 90.000,E1 282.827} C_DIS
LIN {X -0.202,Y -456.627,Z 899.566,A 0.000,B 0.000,C 90.000,E1 281.827} C_DIS
LIN {X -0.098,Y -464.474,Z 899.560,A 0.000,B 0.000,C 90.000,E1 280.782} C_DIS
LIN {X -0.034,Y -473.664,Z 899.553,A 0.000,B 0.000,C 90.000,E1 279.500} C_DIS
LIN {X -0.060,Y -478.627,Z 899.549,A 0.000,B 0.000,C 90.000,E1 278.746} C_DIS
LIN {X -0.039,Y -482.784,Z 899.544,A 0.000,B 0.000,C 90.000,E1 277.992} C_DIS
LIN {X 0.015,Y -486.265,Z 899.540,A 0.000,B 0.000,C 90.000,E1 277.239} C_DIS
LIN {X 0.211,Y -488.173,Z 899.537,A 0.000,B 0.000,C 90.000,E1 276.720} C_DIS
LIN {X -0.074,Y -489.725,Z 899.535,A 0.000,B 0.000,C 90.000,E1 276.258} C_DIS
LIN {X 0.140,Y -490.977,Z 899.532,A 0.000,B 0.000,C 90.000,E1 275.739} C_DIS
LIN {X -0.128,Y -491.797,Z 899.529,A 0.000,B 0.000,C 90.000,E1 275.277} C_DIS
LIN {X 0.098,Y -492.231,Z 899.526,A 0.000,B 0.000,C 90.000,E1 274.759} C_DIS
LIN {X -0.199,Y -492.299,Z 899.524,A 0.000,B 0.000,C 90.000,E1 274.302} C_DIS
LIN {X 0.034,Y -491.955,Z 899.521,A 0.000,B 0.000,C 90.000,E1 273.784} C_DIS
LIN {X -0.254,Y -491.101,Z 899.518,A 0.000,B 0.000,C 90.000,E1 273.326} C_DIS
LIN {X -0.026,Y -489.779,Z 899.516,A 0.000,B 0.000,C 90.000,E1 272.808} C_DIS
LIN {X 0.170,Y -487.945,Z 899.513,A 0.000,B 0.000,C 90.000,E1 272.293} C_DIS
LIN {X -0.124,Y -485.505,Z 899.510,A 0.000,B 0.000,C 90.000,E1 271.835} C_DIS
LIN {X 0.064,Y -482.389,Z 899.507,A 0.000,B 0.000,C 90.000,E1 271.318} C_DIS
LIN {X 0.220,Y -478.450,Z 899.505,A 0.000,B 0.000,C 90.000,E1 270.802} C_DIS
LIN {X -0.120,Y -473.491,Z 899.502,A 0.000,B 0.000,C 90.000,E1 270.344} C_DIS
LIN {X 0.131,Y -467.658,Z 899.499,A 0.000,B 0.000,C 90.000,E1 269.828} C_DIS
LIN {X -0.056,Y -461.534,Z 899.497,A 0.000,B 0.000,C 90.000,E1 269.427} C_DIS
LIN {X 0.199,Y -455.184,Z 899.495,A 0.000,B 0.000,C 90.000,E1 269.026} C_DIS
LIN {X -0.090,Y -448.430,Z 899.493,A 0.000,B 0.000,C 90.000,E1 268.740} C_DIS
LIN {X -0.007,Y -441.214,Z 899.491,A 0.000,B 0.000,C 90.000,E1 268.453} C_DIS
LIN {X 0.054,Y -433.993,Z 899.490,A 0.000,B 0.000,C 90.000,E1 268.224} C_DIS
LIN {X 0.006,Y -426.123,Z 899.489,A 0.000,B 0.000,C 90.000,E1 268.051} C_DIS
LIN {X -0.140,Y -417.321,Z 899.488,A 0.000,B 0.000,C 90.000,E1 267.936} C_DIS
LIN {X 0.132,Y -406.331,Z 899.488,A 0.000,B 0.000,C 90.000,E1 267.822} C_DIS
LIN {X 0.040,Y -181.098,Z 899.488,A 0.000,B 0.000,C 90.000,E1 267.822} C_DIS
LIN {X 0.022,Y -180.852,Z 899.472,A 0.000,B 0.000,C 90.000,E1 264.951} C_DIS
LIN {X -0.072,Y -178.962,Z 899.444,A 0.000,B 0.000,C 90.000,E1 259.916} C_DIS
LIN {X -0.004,Y -177.370,Z 899.430,A 0.000,B 0.000,C 90.000,E1 257.353} C_DIS
LIN {X -0.078,Y -175.545,Z 899.411,A 0.000,B 0.000,C 90.000,E1 253.976} C_DIS
LIN {X -0.070,Y -172.277,Z 899.387,A 0.000,B 0.000,C 90.000,E1 249.699} C_DIS
LIN {X -0.030,Y -171.756,Z 899.382,A 0.000,B 0.000,C 90.000,E1 248.827} C_DIS
LIN {X -0.013,Y -167.355,Z 899.354,A 0.000,B 0.000,C 90.000,E1 243.640} C_DIS
LIN {X 0.069,Y -166.744,Z 899.349,A 0.000,B 0.000,C 90.000,E1 242.743} C_DIS
LIN {X -0.019,Y -162.723,Z 899.324,A 0.000,B 0.000,C 90.000,E1 238.408} C_DIS
LIN {X 0.042,Y -161.415,Z 899.315,A 0.000,B 0.000,C 90.000,E1 236.628} C_DIS
LIN {X 0.083,Y -157.407,Z 899.290,A 0.000,B 0.000,C 90.000,E1 232.190} C_DIS
LIN {X 0.016,Y -155.407,Z 899.275,A 0.000,B 0.000,C 90.000,E1 229.542} C_DIS
LIN {X -0.052,Y -151.737,Z 899.250,A 0.000,B 0.000,C 90.000,E1 225.081} C_DIS
LIN {X -0.041,Y -149.933,Z 899.235,A 0.000,B 0.000,C 90.000,E1 222.366} C_DIS
LIN {X -0.012,Y -146.782,Z 899.210,A 0.000,B 0.000,C 90.000,E1 217.810} C_DIS
LIN {X 0.091,Y -145.354,Z 899.195,A 0.000,B 0.000,C 90.000,E1 215.025} C_DIS
LIN {X 0.006,Y -142.425,Z 899.164,A 0.000,B 0.000,C 90.000,E1 209.539} C_DIS
LIN {X 0.055,Y -141.413,Z 899.149,A 0.000,B 0.000,C 90.000,E1 206.744} C_DIS
LIN {X 0.043,Y -139.359,Z 899.113,A 0.000,B 0.000,C 90.000,E1 200.248} C_DIS
LIN {X 0.030,Y -138.802,Z 899.097,A 0.000,B 0.000,C 90.000,E1 197.457} C_DIS
LIN {X -0.052,Y -138.349,Z 899.056,A 0.000,B 0.000,C 90.000,E1 190.018} C_DIS
LIN {X -0.037,Y -139.366,Z 899.009,A 0.000,B 0.000,C 90.000,E1 181.604} C_DIS
LIN {X 0.016,Y -141.252,Z 898.973,A 0.000,B 0.000,C 90.000,E1 175.065} C_DIS
LIN {X -0.025,Y -142.621,Z 898.957,A 0.000,B 0.000,C 90.000,E1 172.299} C_DIS
LIN {X 0.069,Y -144.940,Z 898.932,A 0.000,B 0.000,C 90.000,E1 167.645} C_DIS
LIN {X 0.061,Y -147.569,Z 898.911,A 0.000,B 0.000,C 90.000,E1 163.976} C_DIS
LIN {X -0.050,Y -150.177,Z 898.891,A 0.000,B 0.000,C 90.000,E1 160.369} C_DIS
LIN {X -0.042,Y -153.555,Z 898.871,A 0.000,B 0.000,C 90.000,E1 156.741} C_DIS
LIN {X 0.009,Y -156.971,Z 898.851,A 0.000,B 0.000,C 90.000,E1 153.127} C_DIS
LIN {X 0.084,Y -161.081,Z 898.831,A 0.000,B 0.000,C 90.000,E1 149.537} C_DIS
LIN {X 0.029,Y -163.188,Z 898.821,A 0.000,B 0.000,C 90.000,E1 147.788} C_DIS
LIN {X 0.035,Y -167.611,Z 898.802,A 0.000,B 0.000,C 90.000,E1 144.276} C_DIS
LIN {X -0.056,Y -171.438,Z 898.787,A 0.000,B 0.000,C 90.000,E1 141.698} C_DIS
LIN {X -0.019,Y -176.359,Z 898.768,A 0.000,B 0.000,C 90.000,E1 138.243} C_DIS
LIN {X 0.105,Y -180.651,Z 898.754,A 0.000,B 0.000,C 90.000,E1 135.648} C_DIS
LIN {X -0.038,Y -186.053,Z 898.735,A 0.000,B 0.000,C 90.000,E1 132.324} C_DIS
LIN {X 0.025,Y -190.689,Z 898.721,A 0.000,B 0.000,C 90.000,E1 129.806} C_DIS
LIN {X -0.074,Y -193.473,Z 898.712,A 0.000,B 0.000,C 90.000,E1 128.177} C_DIS
LIN {X -0.149,Y -294.713,Z 898.712,A 0.000,B 0.000,C 90.000,E1 128.177} C_DIS
LIN {X -0.019,Y -297.667,Z 898.712,A 0.000,B 0.000,C 90.000,E1 128.096} C_DIS
LIN {X 0.074,Y -301.327,Z 898.711,A 0.000,B 0.000,C 90.000,E1 127.890} C_DIS
LIN {X -0.071,Y -303.570,Z 898.710,A 0.000,B 0.000,C 90.000,E1 127.729} C_DIS
LIN {X -0.124,Y -306.689,Z 898.707,A 0.000,B 0.000,C 90.000,E1 127.363} C_DIS
LIN {X -0.085,Y -308.628,Z 898.706,A 0.000,B 0.000,C 90.000,E1 127.030} C_DIS
LIN {X 0.142,Y -310.137,Z 898.704,A 0.000,B 0.000,C 90.000,E1 126.664} C_DIS
LIN {X 0.151,Y -312.299,Z 898.700,A 0.000,B 0.000,C 90.000,E1 126.011} C_DIS
LIN {X -0.088,Y -322.587,Z 898.682,A 0.000,B 0.000,C 90.000,E1 122.832} C_DIS
LIN {X -0.182,Y -333.178,Z 898.667,A 0.000,B 0.000,C 90.000,E1 120.001} C_DIS
LIN {X -0.029,Y -345.135,Z 898.651,A 0.000,B 0.000,C 90.000,E1 117.180} C_DIS
LIN {X -0.154,Y -358.558,Z 898.636,A 0.000,B 0.000,C 90.000,E1 114.463} C_DIS
LIN {X -0.136,Y -371.821,Z 898.623,A 0.000,B 0.000,C 90.000,E1 112.078} C_DIS
LIN {X -0.208,Y -386.434,Z 898.610,A 0.000,B 0.000,C 90.000,E1 109.758} C_DIS
LIN {X -0.037,Y -402.500,Z 898.597,A 0.000,B 0.000,C 90.000,E1 107.457} C_DIS
LIN {X -0.095,Y -420.137,Z 898.585,A 0.000,B 0.000,C 90.000,E1 105.245} C_DIS
LIN {X 0.109,Y -439.419,Z 898.573,A 0.000,B 0.000,C 90.000,E1 103.063} C_DIS
LIN {X -0.025,Y -459.602,Z 898.562,A 0.000,B 0.000,C 90.000,E1 101.074} C_DIS
LIN {X -0.050,Y -467.290,Z 898.558,A 0.000,B 0.000,C 90.000,E1 100.366} C_DIS
LIN {X -0.132,Y -469.343,Z 898.556,A 0.000,B 0.000,C 90.000,E1 100.141} C_DIS
LIN {X -0.131,Y -470.902,Z 898.555,A 0.000,B 0.000,C 90.000,E1 99.905} C_DIS
LIN {X 0.187,Y -472.174,Z 898.554,A 0.000,B 0.000,C 90.000,E1 99.613} C_DIS
LIN {X 0.039,Y -473.111,Z 898.552,A 0.000,B 0.000,C 90.000,E1 99.378} C_DIS
LIN {X 0.149,Y -474.145,Z 898.549,A 0.000,B 0.000,C 90.000,E1 98.859} C_DIS
LIN {X -0.201,Y -474.193,Z 898.547,A 0.000,B 0.000,C 90.000,E1 98.398} C_DIS
LIN {X -0.009,Y -473.266,Z 898.544,A 0.000,B 0.000,C 90.000,E1 97.871} C_DIS
LIN {X 0.115,Y -471.212,Z 898.541,A 0.000,B 0.000,C 90.000,E1 97.352} C_DIS
LIN {X -0.185,Y -453.746,Z 898.525,A 0.000,B 0.000,C 90.000,E1 94.588} C_DIS
LIN {X -0.039,Y -443.091,Z 898.515,A 0.000,B 0.000,C 90.000,E1 92.751} C_DIS
LIN {X 0.141,Y -433.564,Z 898.506,A 0.000,B 0.000,C 90.000,E1 91.146} C_DIS
LIN {X 0.144,Y -423.893,Z 898.498,A 0.000,B 0.000,C 90.000,E1 89.542} C_DIS
LIN {X -0.159,Y -409.412,Z 898.484,A 0.000,B 0.000,C 90.000,E1 87.135} C_DIS
LIN {X -0.052,Y -398.232,Z 898.473,A 0.000,B 0.000,C 90.000,E1 85.179} C_DIS
LIN {X -0.131,Y -385.533,Z 898.461,A 0.000,B 0.000,C 90.000,E1 82.932} C_DIS
LIN {X -0.057,Y -376.010,Z 898.451,A 0.000,B 0.000,C 90.000,E1 81.197} C_DIS
LIN {X -0.102,Y -366.399,Z 898.441,A 0.000,B 0.000,C 90.000,E1 79.454} C_DIS
LIN {X 0.051,Y -355.023,Z 898.430,A 0.000,B 0.000,C 90.000,E1 77.353} C_DIS
LIN {X 0.116,Y -343.613,Z 898.418,A 0.000,B 0.000,C 90.000,E1 75.227} C_DIS
LIN {X -0.153,Y -327.788,Z 898.401,A 0.000,B 0.000,C 90.000,E1 72.181} C_DIS
LIN {X -0.091,Y -314.371,Z 898.385,A 0.000,B 0.000,C 90.000,E1 69.316} C_DIS
LIN {X 0.009,Y -305.544,Z 898.374,A 0.000,B 0.000,C 90.000,E1 67.358} C_DIS
LIN {X 0.045,Y -293.914,Z 898.360,A 0.000,B 0.000,C 90.000,E1 64.717} C_DIS
LIN {X -0.152,Y -285.116,Z 898.348,A 0.000,B 0.000,C 90.000,E1 62.743} C_DIS
LIN {X -0.049,Y -274.714,Z 898.335,A 0.000,B 0.000,C 90.000,E1 60.333} C_DIS
LIN {X 0.055,Y -261.738,Z 898.318,A 0.000,B 0.000,C 90.000,E1 57.168} C_DIS
LIN {X -0.124,Y -249.789,Z 898.300,A 0.000,B 0.000,C 90.000,E1 53.989} C_DIS
LIN {X -0.031,Y -241.444,Z 898.286,A 0.000,B 0.000,C 90.000,E1 51.412} C_DIS
LIN {X -0.093,Y -231.666,Z 898.267,A 0.000,B 0.000,C 90.000,E1 48.081} C_DIS
LIN {X -0.011,Y -221.787,Z 898.246,A 0.000,B 0.000,C 90.000,E1 44.271} C_DIS
LIN {X 0.118,Y -214.310,Z 898.229,A 0.000,B 0.000,C 90.000,E1 41.148} C_DIS
LIN {X 0.097,Y -207.356,Z 898.211,A 0.000,B 0.000,C 90.000,E1 38.016} C_DIS
LIN {X -0.057,Y -199.374,Z 898.189,A 0.000,B 0.000,C 90.000,E1 34.072} C_DIS
LIN {X 0.064,Y -193.511,Z 898.171,A 0.000,B 0.000,C 90.000,E1 30.797} C_DIS
LIN {X 0.068,Y -188.309,Z 898.153,A 0.000,B 0.000,C 90.000,E1 27.513} C_DIS
LIN {X 0.023,Y -183.715,Z 898.135,A 0.000,B 0.000,C 90.000,E1 24.207} C_DIS
LIN {X 0.074,Y -178.912,Z 898.111,A 0.000,B 0.000,C 90.000,E1 19.993} C_DIS
LIN {X -0.041,Y -175.248,Z 898.088,A 0.000,B 0.000,C 90.000,E1 15.788} C_DIS
LIN {X -0.053,Y -172.314,Z 898.059,A 0.000,B 0.000,C 90.000,E1 10.658} C_DIS
LIN {X -0.047,Y -172.925,Z 897.964,A 0.000,B 0.000,C 90.000,E1 353.514} C_DIS
LIN {X -0.025,Y -175.549,Z 897.940,A 0.000,B 0.000,C 90.000,E1 349.218} C_DIS
LIN {X 0.044,Y -179.122,Z 897.916,A 0.000,B 0.000,C 90.000,E1 344.936} C_DIS
LIN {X -0.050,Y -182.854,Z 897.898,A 0.000,B 0.000,C 90.000,E1 341.583} C_DIS
LIN {X -0.051,Y -187.414,Z 897.879,A 0.000,B 0.000,C 90.000,E1 338.230} C_DIS
LIN {X -0.077,Y -192.757,Z 897.861,A 0.000,B 0.000,C 90.000,E1 334.921} C_DIS
LIN {X 0.047,Y -200.339,Z 897.838,A 0.000,B 0.000,C 90.000,E1 330.795} C_DIS
LIN {X 0.018,Y -206.844,Z 897.820,A 0.000,B 0.000,C 90.000,E1 327.582} C_DIS
LIN {X 0.031,Y -213.843,Z 897.802,A 0.000,B 0.000,C 90.000,E1 324.402} C_DIS
LIN {X 0.043,Y -222.327,Z 897.783,A 0.000,B 0.000,C 90.000,E1 320.884} C_DIS
LIN {X -0.037,Y -230.606,Z 897.766,A 0.000,B 0.000,C 90.000,E1 317.838} C_DIS
LIN {X 0.047,Y -241.037,Z 897.747,A 0.000,B 0.000,C 90.000,E1 314.433} C_DIS
LIN {X -0.079,Y -251.375,Z 897.731,A 0.000,B 0.000,C 90.000,E1 311.515} C_DIS
LIN {X -0.008,Y -264.331,Z 897.713,A 0.000,B 0.000,C 90.000,E1 308.257} C_DIS
LIN {X -0.044,Y -278.612,Z 897.695,A 0.000,B 0.000,C 90.000,E1 305.105} C_DIS
LIN {X 0.092,Y -294.366,Z 897.678,A 0.000,B 0.000,C 90.000,E1 302.005} C_DIS
LIN {X 0.033,Y -309.578,Z 897.663,A 0.000,B 0.000,C 90.000,E1 299.361} C_DIS
LIN {X -0.151,Y -324.265,Z 897.651,A 0.000,B 0.000,C 90.000,E1 297.129} C_DIS
LIN {X 0.002,Y -337.933,Z 897.640,A 0.000,B 0.000,C 90.000,E1 295.207} C_DIS
LIN {X 0.034,Y -360.264,Z 897.625,A 0.000,B 0.000,C 90.000,E1 292.461} C_DIS
LIN {X -0.099,Y -380.935,Z 897.612,A 0.000,B 0.000,C 90.000,E1 290.174} C_DIS
LIN {X -0.067,Y -399.172,Z 897.601,A 0.000,B 0.000,C 90.000,E1 288.236} C_DIS
LIN {X -0.155,Y -411.827,Z 897.594,A 0.000,B 0.000,C 90.000,E1 286.913} C_DIS
LIN {X -0.014,Y -424.400,Z 897.586,A 0.000,B 0.000,C 90.000,E1 285.552} C_DIS
LIN {X -0.078,Y -434.122,Z 897.580,A 0.000,B 0.000,C 90.000,E1 284.481} C_DIS
LIN {X -0.045,Y -443.403,Z 897.574,A 0.000,B 0.000,C 90.000,E1 283.411} C_DIS
LIN {X -0.007,Y -452.117,Z 897.569,A 0.000,B 0.000,C 90.000,E1 282.355} C_DIS
LIN {X 0.135,Y -460.357,Z 897.563,A 0.000,B 0.000,C 90.000,E1 281.299} C_DIS
LIN {X 0.136,Y -469.784,Z 897.556,A 0.000,B 0.000,C 90.000,E1 280.018} C_DIS
LIN {X 0.074,Y -475.137,Z 897.552,A 0.000,B 0.000,C 90.000,E1 279.265} C_DIS
LIN {X 0.065,Y -479.849,Z 897.547,A 0.000,B 0.000,C 90.000,E1 278.511} C_DIS
LIN {X 0.092,Y -483.845,Z 897.543,A 0.000,B 0.000,C 90.000,E1 277.757} C_DIS
LIN {X -0.212,Y -486.120,Z 897.540,A 0.000,B 0.000,C 90.000,E1 277.296} C_DIS
LIN {X -0.019,Y -488.052,Z 897.538,A 0.000,B 0.000,C 90.000,E1 276.777} C_DIS
LIN {X 0.183,Y -489.654,Z 897.535,A 0.000,B 0.000,C 90.000,E1 276.258} C_DIS
LIN {X -0.093,Y -490.911,Z 897.532,A 0.000,B 0.000,C 90.000,E1 275.796} C_DIS
LIN {X 0.128,Y -491.770,Z 897.529,A 0.000,B 0.000,C 90.000,E1 275.277} C_DIS
LIN {X -0.177,Y -492.252,Z 897.527,A 0.000,B 0.000,C 90.000,E1 274.821} C_DIS
LIN {X 0.056,Y -492.361,Z 897.524,A 0.000,B 0.000,C 90.000,E1 274.302} C_DIS
LIN {X -0.201,Y -492.031,Z 897.521,A 0.000,B 0.000,C 90.000,E1 273.841} C_DIS
LIN {X 0.001,Y -491.232,Z 897.518,A 0.000,B 0.000,C 90.000,E1 273.326} C_DIS
LIN {X 0.228,Y -489.978,Z 897.516,A 0.000,B 0.000,C 90.000,E1 272.808} C_DIS
LIN {X -0.063,Y -488.167,Z 897.513,A 0.000,B 0.000,C 90.000,E1 272.350} C_DIS
LIN {X 0.130,Y -485.826,Z 897.510,A 0.000,B 0.000,C 90.000,E1 271.835} C_DIS
LIN {X -0.164,Y -482.803,Z 897.508,A 0.000,B 0.000,C 90.000,E1 271.375} C_DIS
LIN {X -0.004,Y -478.979,Z 897.505,A 0.000,B 0.000,C 90.000,E1 270.859} C_DIS
LIN {X 0.135,Y -474.165,Z 897.502,A 0.000,B 0.000,C 90.000,E1 270.344} C_DIS
LIN {X -0.008,Y -471.436,Z 897.501,A 0.000,B 0.000,C 90.000,E1 270.115} C_DIS
LIN {X -0.030,Y -465.548,Z 897.498,A 0.000,B 0.000,C 90.000,E1 269.656} C_DIS
LIN {X -0.054,Y -459.292,Z 897.496,A 0.000,B 0.000,C 90.000,E1 269.255} C_DIS
LIN {X -0.137,Y -452.690,Z 897.494,A 0.000,B 0.000,C 90.000,E1 268.912} C_DIS
LIN {X 0.174,Y -445.767,Z 897.492,A 0.000,B 0.000,C 90.000,E1 268.568} C_DIS
LIN {X -0.013,Y -438.640,Z 897.491,A 0.000,B 0.000,C 90.000,E1 268.339} C_DIS
LIN {X 0.188,Y -431.070,Z 897.490,A 0.000,B 0.000,C 90.000,E1 268.108} C_DIS
LIN {X -0.147,Y -423.119,Z 897.489,A 0.000,B 0.000,C 90.000,E1 267.993} C_DIS
LIN {X -0.143,Y -413.589,Z 897.488,A 0.000,B 0.000,C 90.000,E1 267.879} C_DIS
LIN {X -0.017,Y -406.793,Z 897.488,A 0.000,B 0.000,C 90.000,E1 267.822} C_DIS
LIN {X -0.029,Y -181.095,Z 897.488,A 0.000,B 0.000,C 90.000,E1 267.822} C_DIS
LIN {X -0.030,Y -180.847,Z 897.472,A 0.000,B 0.000,C 90.000,E1 264.951} C_DIS
LIN {X 0.052,Y -178.957,Z 897.444,A 0.000,B 0.000,C 90.000,E1 259.859} C_DIS
LIN {X -0.056,Y -177.360,Z 897.430,A 0.000,B 0.000,C 90.000,E1 257.353} C_DIS
LIN {X 0.040,Y -175.532,Z 897.411,A 0.000,B 0.000,C 90.000,E1 253.921} C_DIS
LIN {X 0.041,Y -172.267,Z 897.387,A 0.000,B 0.000,C 90.000,E1 249.645} C_DIS
LIN {X 0.080,Y -171.745,Z 897.382,A 0.000,B 0.000,C 90.000,E1 248.773} C_DIS
LIN {X -0.062,Y -167.344,Z 897.353,A 0.000,B 0.000,C 90.000,E1 243.640} C_DIS
LIN {X 0.019,Y -166.730,Z 897.349,A 0.000,B 0.000,C 90.000,E1 242.743} C_DIS
LIN {X -0.068,Y -162.710,Z 897.324,A 0.000,B 0.000,C 90.000,E1 238.408} C_DIS
LIN {X -0.005,Y -161.401,Z 897.315,A 0.000,B 0.000,C 90.000,E1 236.628} C_DIS
LIN {X 0.036,Y -157.393,Z 897.290,A 0.000,B 0.000,C 90.000,E1 232.190} C_DIS
LIN {X -0.031,Y -155.391,Z 897.275,A 0.000,B 0.000,C 90.000,E1 229.542} C_DIS
LIN {X 0.009,Y -151.725,Z 897.250,A 0.000,B 0.000,C 90.000,E1 225.040} C_DIS
LIN {X 0.025,Y -149.919,Z 897.235,A 0.000,B 0.000,C 90.000,E1 222.324} C_DIS
LIN {X -0.057,Y -146.772,Z 897.210,A 0.000,B 0.000,C 90.000,E1 217.810} C_DIS
LIN {X 0.046,Y -145.342,Z 897.195,A 0.000,B 0.000,C 90.000,E1 215.025} C_DIS
LIN {X -0.039,Y -142.418,Z 897.164,A 0.000,B 0.000,C 90.000,E1 209.539} C_DIS
LIN {X 0.011,Y -141.405,Z 897.149,A 0.000,B 0.000,C 90.000,E1 206.744} C_DIS
LIN {X -0.002,Y -139.357,Z 897.112,A 0.000,B 0.000,C 90.000,E1 200.248} C_DIS
LIN {X -0.014,Y -138.798,Z 897.097,A 0.000,B 0.000,C 90.000,E1 197.457} C_DIS
LIN {X 0.041,Y -138.348,Z 897.055,A 0.000,B 0.000,C 90.000,E1 189.962} C_DIS
LIN {X 0.058,Y -139.371,Z 897.009,A 0.000,B 0.000,C 90.000,E1 181.547} C_DIS
LIN {X -0.028,Y -141.260,Z 896.973,A 0.000,B 0.000,C 90.000,E1 175.065} C_DIS
LIN {X -0.070,Y -142.628,Z 896.957,A 0.000,B 0.000,C 90.000,E1 172.299} C_DIS
LIN {X 0.023,Y -144.951,Z 896.931,A 0.000,B 0.000,C 90.000,E1 167.645} C_DIS
LIN {X 0.015,Y -147.580,Z 896.911,A 0.000,B 0.000,C 90.000,E1 163.976} C_DIS
LIN {X 0.045,Y -150.192,Z 896.891,A 0.000,B 0.000,C 90.000,E1 160.315} C_DIS
LIN {X -0.089,Y -153.573,Z 896.871,A 0.000,B 0.000,C 90.000,E1 156.741} C_DIS
LIN {X -0.038,Y -156.990,Z 896.851,A 0.000,B 0.000,C 90.000,E1 153.127} C_DIS
LIN {X 0.036,Y -161.104,Z 896.831,A 0.000,B 0.000,C 90.000,E1 149.537} C_DIS
LIN {X -0.019,Y -163.207,Z 896.821,A 0.000,B 0.000,C 90.000,E1 147.788} C_DIS
LIN {X -0.015,Y -167.634,Z 896.802,A 0.000,B 0.000,C 90.000,E1 144.276} C_DIS
LIN {X 0.000,Y -171.460,Z 896.787,A 0.000,B 0.000,C 90.000,E1 141.662} C_DIS
LIN {X -0.069,Y -176.386,Z 896.768,A 0.000,B 0.000,C 90.000,E1 138.243} C_DIS
LIN {X 0.052,Y -180.679,Z 896.754,A 0.000,B 0.000,C 90.000,E1 135.648} C_DIS
LIN {X 0.035,Y -186.081,Z 896.735,A 0.000,B 0.000,C 90.000,E1 132.285} C_DIS
LIN {X -0.028,Y -190.718,Z 896.721,A 0.000,B 0.000,C 90.000,E1 129.806} C_DIS
LIN {X -0.020,Y -193.445,Z 896.712,A 0.000,B 0.000,C 90.000,E1 128.177} C_DIS
LIN {X -0.074,Y -295.164,Z 896.712,A 0.000,B 0.000,C 90.000,E1 128.177} C_DIS
LIN {X 0.085,Y -299.458,Z 896.711,A 0.000,B 0.000,C 90.000,E1 128.016} C_DIS
LIN {X -0.015,Y -302.712,Z 896.710,A 0.000,B 0.000,C 90.000,E1 127.810} C_DIS
LIN {X 0.152,Y -306.383,Z 896.708,A 0.000,B 0.000,C 90.000,E1 127.363} C_DIS
LIN {X 0.024,Y -308.299,Z 896.706,A 0.000,B 0.000,C 90.000,E1 127.076} C_DIS
LIN {X -0.107,Y -309.801,Z 896.704,A 0.000,B 0.000,C 90.000,E1 126.790} C_DIS
LIN {X -0.072,Y -311.050,Z 896.702,A 0.000,B 0.000,C 90.000,E1 126.457} C_DIS
LIN {X 0.082,Y -322.296,Z 896.683,A 0.000,B 0.000,C 90.000,E1 122.880} C_DIS
LIN {X -0.023,Y -332.850,Z 896.667,A 0.000,B 0.000,C 90.000,E1 120.050} C_DIS
LIN {X -0.041,Y -344.769,Z 896.651,A 0.000,B 0.000,C 90.000,E1 117.257} C_DIS
LIN {X -0.020,Y -358.150,Z 896.636,A 0.000,B 0.000,C 90.000,E1 114.515} C_DIS
LIN {X -0.154,Y -371.373,Z 896.623,A 0.000,B 0.000,C 90.000,E1 112.153} C_DIS
LIN {X -0.097,Y -385.943,Z 896.610,A 0.000,B 0.000,C 90.000,E1 109.812} C_DIS
LIN {X 0.060,Y -401.963,Z 896.597,A 0.000,B 0.000,C 90.000,E1 107.511} C_DIS
LIN {X -0.011,Y -419.550,Z 896.585,A 0.000,B 0.000,C 90.000,E1 105.300} C_DIS
LIN {X 0.166,Y -438.792,Z 896.573,A 0.000,B 0.000,C 90.000,E1 103.119} C_DIS
LIN {X -0.012,Y -458.957,Z 896.562,A 0.000,B 0.000,C 90.000,E1 101.130} C_DIS
LIN {X -0.052,Y -466.675,Z 896.558,A 0.000,B 0.000,C 90.000,E1 100.423} C_DIS
LIN {X -0.124,Y -468.872,Z 896.557,A 0.000,B 0.000,C 90.000,E1 100.197} C_DIS
LIN {X -0.112,Y -470.532,Z 896.555,A 0.000,B 0.000,C 90.000,E1 99.962} C_DIS
LIN {X 0.205,Y -471.898,Z 896.554,A 0.000,B 0.000,C 90.000,E1 99.670} C_DIS
LIN {X -0.022,Y -472.911,Z 896.552,A 0.000,B 0.000,C 90.000,E1 99.443} C_DIS
LIN {X 0.164,Y -474.072,Z 896.550,A 0.000,B 0.000,C 90.000,E1 98.916} C_DIS
LIN {X -0.188,Y -474.236,Z 896.547,A 0.000,B 0.000,C 90.000,E1 98.454} C_DIS
LIN {X -0.062,Y -473.431,Z 896.544,A 0.000,B 0.000,C 90.000,E1 97.936} C_DIS
LIN {X 0.126,Y -471.528,Z 896.541,A 0.000,B 0.000,C 90.000,E1 97.409} C_DIS
LIN {X 0.037,Y -466.758,Z 896.537,A 0.000,B 0.000,C 90.000,E1 96.663} C_DIS
LIN {X 0.019,Y -446.539,Z 896.518,A 0.000,B 0.000,C 90.000,E1 93.326} C_DIS
LIN {X 0.091,Y -438.774,Z 896.511,A 0.000,B 0.000,C 90.000,E1 92.007} C_DIS
LIN {X -0.088,Y -427.580,Z 896.501,A 0.000,B 0.000,C 90.000,E1 90.172} C_DIS
LIN {X 0.036,Y -414.604,Z 896.489,A 0.000,B 0.000,C 90.000,E1 87.993} C_DIS
LIN {X 0.191,Y -403.417,Z 896.478,A 0.000,B 0.000,C 90.000,E1 86.045} C_DIS
LIN {X -0.173,Y -390.643,Z 896.466,A 0.000,B 0.000,C 90.000,E1 83.856} C_DIS
LIN {X -0.029,Y -379.573,Z 896.455,A 0.000,B 0.000,C 90.000,E1 81.837} C_DIS
LIN {X -0.019,Y -368.373,Z 896.443,A 0.000,B 0.000,C 90.000,E1 79.803} C_DIS
LIN {X 0.184,Y -357.068,Z 896.432,A 0.000,B 0.000,C 90.000,E1 77.701} C_DIS
LIN {X -0.135,Y -345.695,Z 896.420,A 0.000,B 0.000,C 90.000,E1 75.644} C_DIS
LIN {X 0.010,Y -331.328,Z 896.405,A 0.000,B 0.000,C 90.000,E1 72.851} C_DIS
LIN {X -0.014,Y -316.294,Z 896.387,A 0.000,B 0.000,C 90.000,E1 69.699} C_DIS
LIN {X -0.169,Y -307.466,Z 896.376,A 0.000,B 0.000,C 90.000,E1 67.794} C_DIS
LIN {X -0.080,Y -295.811,Z 896.362,A 0.000,B 0.000,C 90.000,E1 65.153} C_DIS
LIN {X -0.001,Y -285.611,Z 896.349,A 0.000,B 0.000,C 90.000,E1 62.794} C_DIS
LIN {X -0.023,Y -275.213,Z 896.336,A 0.000,B 0.000,C 90.000,E1 60.411} C_DIS
LIN {X 0.089,Y -262.250,Z 896.318,A 0.000,B 0.000,C 90.000,E1 57.248} C_DIS
LIN {X -0.082,Y -250.317,Z 896.300,A 0.000,B 0.000,C 90.000,E1 54.069} C_DIS
LIN {X 0.020,Y -241.970,Z 896.286,A 0.000,B 0.000,C 90.000,E1 51.492} C_DIS
LIN {X -0.025,Y -232.195,Z 896.268,A 0.000,B 0.000,C 90.000,E1 48.162} C_DIS
LIN {X 0.070,Y -222.311,Z 896.247,A 0.000,B 0.000,C 90.000,E1 44.352} C_DIS
LIN {X -0.093,Y -214.841,Z 896.229,A 0.000,B 0.000,C 90.000,E1 41.310} C_DIS
LIN {X -0.091,Y -207.871,Z 896.212,A 0.000,B 0.000,C 90.000,E1 38.177} C_DIS
LIN {X -0.105,Y -199.847,Z 896.190,A 0.000,B 0.000,C 90.000,E1 34.199} C_DIS
LIN {X 0.026,Y -193.978,Z 896.172,A 0.000,B 0.000,C 90.000,E1 30.924} C_DIS
LIN {X 0.041,Y -188.729,Z 896.154,A 0.000,B 0.000,C 90.000,E1 27.641} C_DIS
LIN {X 0.007,Y -184.124,Z 896.135,A 0.000,B 0.000,C 90.000,E1 24.335} C_DIS
LIN {X 0.074,Y -179.298,Z 896.112,A 0.000,B 0.000,C 90.000,E1 20.120} C_DIS
LIN {X 0.022,Y -175.606,Z 896.088,A 0.000,B 0.000,C 90.000,E1 15.898} C_DIS
LIN {X -0.018,Y -172.621,Z 896.060,A 0.000,B 0.000,C 90.000,E1 10.782} C_DIS
LIN {X -0.035,Y -173.207,Z 895.964,A 0.000,B 0.000,C 90.000,E1 353.514} C_DIS
LIN {X -0.005,Y -175.839,Z 895.940,A 0.000,B 0.000,C 90.000,E1 349.218} C_DIS
LIN {X 0.074,Y -179.431,Z 895.916,A 0.000,B 0.000,C 90.000,E1 344.936} C_DIS
LIN {X -0.012,Y -183.187,Z 895.898,A 0.000,B 0.000,C 90.000,E1 341.583} C_DIS
LIN {X -0.003,Y -187.763,Z 895.879,A 0.000,B 0.000,C 90.000,E1 338.230} C_DIS
LIN {X -0.019,Y -193.112,Z 895.861,A 0.000,B 0.000,C 90.000,E1 334.921} C_DIS
LIN {X -0.001,Y -199.131,Z 895.842,A 0.000,B 0.000,C 90.000,E1 331.641} C_DIS
LIN {X 0.010,Y -205.493,Z 895.825,A 0.000,B 0.000,C 90.000,E1 328.408} C_DIS
LIN {X 0.124,Y -214.156,Z 895.802,A 0.000,B 0.000,C 90.000,E1 324.402} C_DIS
LIN {X -0.023,Y -222.623,Z 895.783,A 0.000,B 0.000,C 90.000,E1 320.928} C_DIS
LIN {X 0.073,Y -230.873,Z 895.766,A 0.000,B 0.000,C 90.000,E1 317.838} C_DIS
LIN {X -0.001,Y -241.298,Z 895.747,A 0.000,B 0.000,C 90.000,E1 314.474} C_DIS
LIN {X 0.057,Y -251.606,Z 895.731,A 0.000,B 0.000,C 90.000,E1 311.515} C_DIS
LIN {X -0.066,Y -264.541,Z 895.713,A 0.000,B 0.000,C 90.000,E1 308.302} C_DIS
LIN {X 0.118,Y -278.750,Z 895.695,A 0.000,B 0.000,C 90.000,E1 305.105} C_DIS
LIN {X 0.018,Y -294.388,Z 895.678,A 0.000,B 0.000,C 90.000,E1 302.054} C_DIS
LIN {X -0.052,Y -309.522,Z 895.663,A 0.000,B 0.000,C 90.000,E1 299.411} C_DIS
LIN {X -0.021,Y -326.282,Z 895.649,A 0.000,B 0.000,C 90.000,E1 296.821} C_DIS
LIN {X -0.128,Y -340.093,Z 895.638,A 0.000,B 0.000,C 90.000,E1 294.951} C_DIS
LIN {X 0.033,Y -359.743,Z 895.625,A 0.000,B 0.000,C 90.000,E1 292.514} C_DIS
LIN {X 0.142,Y -382.641,Z 895.611,A 0.000,B 0.000,C 90.000,E1 289.939} C_DIS
LIN {X 0.005,Y -400.604,Z 895.600,A 0.000,B 0.000,C 90.000,E1 288.055} C_DIS
LIN {X 0.223,Y -413.393,Z 895.593,A 0.000,B 0.000,C 90.000,E1 286.677} C_DIS
LIN {X 0.185,Y -423.482,Z 895.587,A 0.000,B 0.000,C 90.000,E1 285.607} C_DIS
LIN {X 0.127,Y -433.249,Z 895.581,A 0.000,B 0.000,C 90.000,E1 284.537} C_DIS
LIN {X 0.049,Y -442.586,Z 895.575,A 0.000,B 0.000,C 90.000,E1 283.480} C_DIS
LIN {X 0.182,Y -451.382,Z 895.569,A 0.000,B 0.000,C 90.000,E1 282.411} C_DIS
LIN {X -0.224,Y -459.697,Z 895.563,A 0.000,B 0.000,C 90.000,E1 281.422} C_DIS
LIN {X 0.005,Y -467.340,Z 895.558,A 0.000,B 0.000,C 90.000,E1 280.366} C_DIS
LIN {X 0.245,Y -474.565,Z 895.552,A 0.000,B 0.000,C 90.000,E1 279.321} C_DIS
LIN {X 0.231,Y -479.331,Z 895.548,A 0.000,B 0.000,C 90.000,E1 278.568} C_DIS
LIN {X 0.254,Y -483.435,Z 895.544,A 0.000,B 0.000,C 90.000,E1 277.814} C_DIS
LIN {X -0.051,Y -485.772,Z 895.541,A 0.000,B 0.000,C 90.000,E1 277.352} C_DIS
LIN {X 0.139,Y -487.781,Z 895.538,A 0.000,B 0.000,C 90.000,E1 276.834} C_DIS
LIN {X -0.149,Y -489.432,Z 895.535,A 0.000,B 0.000,C 90.000,E1 276.372} C_DIS
LIN {X 0.061,Y -490.725,Z 895.533,A 0.000,B 0.000,C 90.000,E1 275.853} C_DIS
LIN {X -0.209,Y -491.679,Z 895.530,A 0.000,B 0.000,C 90.000,E1 275.391} C_DIS
LIN {X -0.027,Y -492.242,Z 895.527,A 0.000,B 0.000,C 90.000,E1 274.878} C_DIS
LIN {X 0.207,Y -492.394,Z 895.524,A 0.000,B 0.000,C 90.000,E1 274.359} C_DIS
LIN {X -0.051,Y -492.128,Z 895.522,A 0.000,B 0.000,C 90.000,E1 273.898} C_DIS
LIN {X 0.150,Y -491.438,Z 895.519,A 0.000,B 0.000,C 90.000,E1 273.383} C_DIS
LIN {X -0.112,Y -490.237,Z 895.516,A 0.000,B 0.000,C 90.000,E1 272.922} C_DIS
LIN {X 0.087,Y -488.585,Z 895.513,A 0.000,B 0.000,C 90.000,E1 272.407} C_DIS
LIN {X -0.205,Y -486.349,Z 895.511,A 0.000,B 0.000,C 90.000,E1 271.949} C_DIS
LIN {X -0.012,Y -483.471,Z 895.508,A 0.000,B 0.000,C 90.000,E1 271.432} C_DIS
LIN {X -0.170,Y -481.795,Z 895.507,A 0.000,B 0.000,C 90.000,E1 271.203} C_DIS
LIN {X -0.016,Y -477.654,Z 895.504,A 0.000,B 0.000,C 90.000,E1 270.688} C_DIS
LIN {X 0.116,Y -472.598,Z 895.501,A 0.000,B 0.000,C 90.000,E1 270.172} C_DIS
LIN {X -0.010,Y -466.783,Z 895.498,A 0.000,B 0.000,C 90.000,E1 269.714} C_DIS
LIN {X -0.171,Y -460.542,Z 895.496,A 0.000,B 0.000,C 90.000,E1 269.312} C_DIS
LIN {X 0.092,Y -453.901,Z 895.494,A 0.000,B 0.000,C 90.000,E1 268.912} C_DIS
LIN {X -0.117,Y -446.989,Z 895.492,A 0.000,B 0.000,C 90.000,E1 268.625} C_DIS
LIN {X 0.074,Y -439.780,Z 895.491,A 0.000,B 0.000,C 90.000,E1 268.339} C_DIS
LIN {X 0.190,Y -432.160,Z 895.490,A 0.000,B 0.000,C 90.000,E1 268.108} C_DIS
LIN {X 0.203,Y -423.864,Z 895.489,A 0.000,B 0.000,C 90.000,E1 267.936} C_DIS
LIN {X 0.172,Y -414.758,Z 895.488,A 0.000,B 0.000,C 90.000,E1 267.822} C_DIS
LIN {X -0.142,Y -408.021,Z 895.488,A 0.000,B 0.000,C 90.000,E1 267.822} C_DIS
LIN {X -0.086,Y -181.092,Z 895.488,A 0.000,B 0.000,C 90.000,E1 267.822} C_DIS
LIN {X 0.090,Y -180.843,Z 895.472,A 0.000,B 0.000,C 90.000,E1 264.894} C_DIS
LIN {X -0.008,Y -178.951,Z 895.444,A 0.000,B 0.000,C 90.000,E1 259.859} C_DIS
LIN {X 0.009,Y -176.856,Z 895.425,A 0.000,B 0.000,C 90.000,E1 256.464} C_DIS
LIN {X -0.019,Y -175.516,Z 895.411,A 0.000,B 0.000,C 90.000,E1 253.921} C_DIS
LIN {X -0.017,Y -172.254,Z 895.387,A 0.000,B 0.000,C 90.000,E1 249.645} C_DIS
LIN {X 0.022,Y -171.733,Z 895.382,A 0.000,B 0.000,C 90.000,E1 248.773} C_DIS
LIN {X 0.031,Y -167.330,Z 895.353,A 0.000,B 0.000,C 90.000,E1 243.589} C_DIS
LIN {X -0.038,Y -166.714,Z 895.349,A 0.000,B 0.000,C 90.000,E1 242.743} C_DIS
LIN {X 0.100,Y -162.694,Z 895.324,A 0.000,B 0.000,C 90.000,E1 238.329} C_DIS
LIN {X -0.061,Y -161.385,Z 895.314,A 0.000,B 0.000,C 90.000,E1 236.628} C_DIS
LIN {X -0.019,Y -157.378,Z 895.290,A 0.000,B 0.000,C 90.000,E1 232.190} C_DIS
LIN {X -0.086,Y -155.371,Z 895.275,A 0.000,B 0.000,C 90.000,E1 229.542} C_DIS
LIN {X 0.062,Y -151.711,Z 895.250,A 0.000,B 0.000,C 90.000,E1 225.000} C_DIS
LIN {X -0.029,Y -149.902,Z 895.235,A 0.000,B 0.000,C 90.000,E1 222.324} C_DIS
LIN {X 0.096,Y -146.761,Z 895.210,A 0.000,B 0.000,C 90.000,E1 217.729} C_DIS
LIN {X -0.006,Y -145.328,Z 895.195,A 0.000,B 0.000,C 90.000,E1 215.025} C_DIS
LIN {X 0.033,Y -142.410,Z 895.164,A 0.000,B 0.000,C 90.000,E1 209.489} C_DIS
LIN {X -0.041,Y -141.395,Z 895.148,A 0.000,B 0.000,C 90.000,E1 206.744} C_DIS
LIN {X -0.053,Y -139.354,Z 895.112,A 0.000,B 0.000,C 90.000,E1 200.248} C_DIS
LIN {X -0.064,Y -138.793,Z 895.097,A 0.000,B 0.000,C 90.000,E1 197.457} C_DIS
LIN {X -0.010,Y -138.347,Z 895.055,A 0.000,B 0.000,C 90.000,E1 189.962} C_DIS
LIN {X 0.007,Y -139.378,Z 895.009,A 0.000,B 0.000,C 90.000,E1 181.547} C_DIS
LIN {X 0.061,Y -141.270,Z 894.972,A 0.000,B 0.000,C 90.000,E1 175.008} C_DIS
LIN {X 0.019,Y -142.636,Z 894.957,A 0.000,B 0.000,C 90.000,E1 172.243} C_DIS
LIN {X -0.029,Y -144.964,Z 894.931,A 0.000,B 0.000,C 90.000,E1 167.645} C_DIS
LIN {X -0.039,Y -147.592,Z 894.911,A 0.000,B 0.000,C 90.000,E1 163.976} C_DIS
LIN {X -0.009,Y -150.209,Z 894.891,A 0.000,B 0.000,C 90.000,E1 160.315} C_DIS
LIN {X 0.058,Y -153.594,Z 894.870,A 0.000,B 0.000,C 90.000,E1 156.666} C_DIS
LIN {X 0.047,Y -157.010,Z 894.851,A 0.000,B 0.000,C 90.000,E1 153.076} C_DIS
LIN {X -0.021,Y -161.129,Z 894.831,A 0.000,B 0.000,C 90.000,E1 149.537} C_DIS
LIN {X -0.076,Y -163.229,Z 894.821,A 0.000,B 0.000,C 90.000,E1 147.788} C_DIS
LIN {X -0.073,Y -167.662,Z 894.801,A 0.000,B 0.000,C 90.000,E1 144.276} C_DIS
LIN {X 0.076,Y -171.486,Z 894.787,A 0.000,B 0.000,C 90.000,E1 141.618} C_DIS
LIN {X 0.120,Y -176.416,Z 894.768,A 0.000,B 0.000,C 90.000,E1 138.162} C_DIS
LIN {X -0.008,Y -180.710,Z 894.754,A 0.000,B 0.000,C 90.000,E1 135.648} C_DIS
LIN {X -0.027,Y -186.114,Z 894.735,A 0.000,B 0.000,C 90.000,E1 132.285} C_DIS
LIN {X 0.031,Y -190.752,Z 894.721,A 0.000,B 0.000,C 90.000,E1 129.769} C_DIS
LIN {X 0.031,Y -193.419,Z 894.712,A 0.000,B 0.000,C 90.000,E1 128.177} C_DIS
LIN {X 0.011,Y -295.166,Z 894.712,A 0.000,B 0.000,C 90.000,E1 128.177} C_DIS
LIN {X 0.159,Y -297.559,Z 894.712,A 0.000,B 0.000,C 90.000,E1 128.096} C_DIS
LIN {X -0.071,Y -300.931,Z 894.711,A 0.000,B 0.000,C 90.000,E1 127.971} C_DIS
LIN {X -0.016,Y -304.434,Z 894.709,A 0.000,B 0.000,C 90.000,E1 127.649} C_DIS
LIN {X -0.136,Y -308.045,Z 894.706,A 0.000,B 0.000,C 90.000,E1 127.156} C_DIS
LIN {X 0.071,Y -309.663,Z 894.704,A 0.000,B 0.000,C 90.000,E1 126.790} C_DIS
LIN {X 0.095,Y -310.934,Z 894.703,A 0.000,B 0.000,C 90.000,E1 126.457} C_DIS
LIN {X -0.191,Y -322.169,Z 894.683,A 0.000,B 0.000,C 90.000,E1 122.959} C_DIS
LIN {X -0.020,Y -332.712,Z 894.667,A 0.000,B 0.000,C 90.000,E1 120.079} C_DIS
LIN {X 0.135,Y -344.612,Z 894.652,A 0.000,B 0.000,C 90.000,E1 117.257} C_DIS
LIN {X 0.154,Y -357.981,Z 894.636,A 0.000,B 0.000,C 90.000,E1 114.515} C_DIS
LIN {X 0.023,Y -371.189,Z 894.623,A 0.000,B 0.000,C 90.000,E1 112.153} C_DIS
LIN {X 0.081,Y -385.742,Z 894.610,A 0.000,B 0.000,C 90.000,E1 109.812} C_DIS
LIN {X 0.120,Y -401.745,Z 894.597,A 0.000,B 0.000,C 90.000,E1 107.528} C_DIS
LIN {X 0.061,Y -419.313,Z 894.585,A 0.000,B 0.000,C 90.000,E1 105.315} C_DIS
LIN {X -0.079,Y -438.539,Z 894.573,A 0.000,B 0.000,C 90.000,E1 103.175} C_DIS
LIN {X 0.161,Y -458.698,Z 894.562,A 0.000,B 0.000,C 90.000,E1 101.130} C_DIS
LIN {X 0.055,Y -466.386,Z 894.558,A 0.000,B 0.000,C 90.000,E1 100.433} C_DIS
LIN {X 0.075,Y -468.651,Z 894.557,A 0.000,B 0.000,C 90.000,E1 100.197} C_DIS
LIN {X -0.062,Y -470.475,Z 894.555,A 0.000,B 0.000,C 90.000,E1 99.962} C_DIS
LIN {X -0.201,Y -471.848,Z 894.554,A 0.000,B 0.000,C 90.000,E1 99.726} C_DIS
LIN {X -0.102,Y -473.595,Z 894.551,A 0.000,B 0.000,C 90.000,E1 99.208} C_DIS
LIN {X 0.080,Y -474.264,Z 894.548,A 0.000,B 0.000,C 90.000,E1 98.681} C_DIS
LIN {X 0.200,Y -473.966,Z 894.545,A 0.000,B 0.000,C 90.000,E1 98.163} C_DIS
LIN {X -0.144,Y -472.660,Z 894.543,A 0.000,B 0.000,C 90.000,E1 97.701} C_DIS
LIN {X 0.183,Y -471.567,Z 894.541,A 0.000,B 0.000,C 90.000,E1 97.409} C_DIS
LIN {X -0.167,Y -468.458,Z 894.539,A 0.000,B 0.000,C 90.000,E1 96.947} C_DIS
LIN {X -0.127,Y -451.125,Z 894.523,A 0.000,B 0.000,C 90.000,E1 94.131} C_DIS
LIN {X -0.215,Y -442.015,Z 894.514,A 0.000,B 0.000,C 90.000,E1 92.579} C_DIS
LIN {X -0.047,Y -432.495,Z 894.505,A 0.000,B 0.000,C 90.000,E1 90.974} C_DIS
LIN {X -0.058,Y -422.811,Z 894.496,A 0.000,B 0.000,C 90.000,E1 89.370} C_DIS
LIN {X -0.052,Y -409.909,Z 894.484,A 0.000,B 0.000,C 90.000,E1 87.192} C_DIS
LIN {X 0.024,Y -398.664,Z 894.474,A 0.000,B 0.000,C 90.000,E1 85.241} C_DIS
LIN {X -0.061,Y -385.956,Z 894.461,A 0.000,B 0.000,C 90.000,E1 82.996} C_DIS
LIN {X 0.066,Y -376.419,Z 894.451,A 0.000,B 0.000,C 90.000,E1 81.254} C_DIS
LIN {X 0.018,Y -365.217,Z 894.440,A 0.000,B 0.000,C 90.000,E1 79.218} C_DIS
LIN {X -0.152,Y -355.527,Z 894.430,A 0.000,B 0.000,C 90.000,E1 77.465} C_DIS
LIN {X -0.070,Y -344.190,Z 894.418,A 0.000,B 0.000,C 90.000,E1 75.338} C_DIS
LIN {X 0.040,Y -329.919,Z 894.403,A 0.000,B 0.000,C 90.000,E1 72.543} C_DIS
LIN {X -0.021,Y -314.976,Z 894.385,A 0.000,B 0.000,C 90.000,E1 69.390} C_DIS
LIN {X 0.083,Y -306.144,Z 894.375,A 0.000,B 0.000,C 90.000,E1 67.433} C_DIS
LIN {X 0.124,Y -294.553,Z 894.360,A 0.000,B 0.000,C 90.000,E1 64.793} C_DIS
LIN {X -0.095,Y -284.307,Z 894.347,A 0.000,B 0.000,C 90.000,E1 62.487} C_DIS
LIN {X -0.013,Y -273.960,Z 894.334,A 0.000,B 0.000,C 90.000,E1 60.078} C_DIS
LIN {X 0.065,Y -261.137,Z 894.316,A 0.000,B 0.000,C 90.000,E1 56.914} C_DIS
LIN {X 0.008,Y -249.345,Z 894.298,A 0.000,B 0.000,C 90.000,E1 53.703} C_DIS
LIN {X -0.101,Y -241.141,Z 894.284,A 0.000,B 0.000,C 90.000,E1 51.170} C_DIS
LIN {X 0.015,Y -231.476,Z 894.266,A 0.000,B 0.000,C 90.000,E1 47.796} C_DIS
LIN {X -0.075,Y -221.684,Z 894.245,A 0.000,B 0.000,C 90.000,E1 44.028} C_DIS
LIN {X -0.122,Y -212.514,Z 894.223,A 0.000,B 0.000,C 90.000,E1 40.172} C_DIS
LIN {X -0.020,Y -205.730,Z 894.206,A 0.000,B 0.000,C 90.000,E1 36.996} C_DIS
LIN {X 0.033,Y -199.400,Z 894.188,A 0.000,B 0.000,C 90.000,E1 33.785} C_DIS
LIN {X 0.048,Y -193.599,Z 894.170,A 0.000,B 0.000,C 90.000,E1 30.541} C_DIS
LIN {X 0.057,Y -188.385,Z 894.152,A 0.000,B 0.000,C 90.000,E1 27.257} C_DIS
LIN {X 0.013,Y -183.893,Z 894.133,A 0.000,B 0.000,C 90.000,E1 23.951} C_DIS
LIN {X 0.005,Y -179.164,Z 894.110,A 0.000,B 0.000,C 90.000,E1 19.758} C_DIS
LIN {X -0.049,Y -175.590,Z 894.086,A 0.000,B 0.000,C 90.000,E1 15.536} C_DIS
LIN {X 0.074,Y -172.708,Z 894.058,A 0.000,B 0.000,C 90.000,E1 10.366} C_DIS
LIN {X -0.023,Y -173.489,Z 893.964,A 0.000,B 0.000,C 90.000,E1 353.514} C_DIS
LIN {X 0.016,Y -176.129,Z 893.940,A 0.000,B 0.000,C 90.000,E1 349.218} C_DIS
LIN {X -0.070,Y -179.741,Z 893.917,A 0.000,B 0.000,C 90.000,E1 344.991} C_DIS
LIN {X 0.027,Y -183.524,Z 893.898,A 0.000,B 0.000,C 90.000,E1 341.583} C_DIS
LIN {X 0.045,Y -188.127,Z 893.879,A 0.000,B 0.000,C 90.000,E1 338.230} C_DIS
LIN {X 0.039,Y -193.470,Z 893.861,A 0.000,B 0.000,C 90.000,E1 334.921} C_DIS
LIN {X 0.068,Y -199.466,Z 893.843,A 0.000,B 0.000,C 90.000,E1 331.641} C_DIS
LIN {X 0.089,Y -205.837,Z 893.825,A 0.000,B 0.000,C 90.000,E1 328.408} C_DIS
LIN {X -0.046,Y -212.679,Z 893.807,A 0.000,B 0.000,C 90.000,E1 325.261} C_DIS
LIN {X 0.012,Y -220.009,Z 893.789,A 0.000,B 0.000,C 90.000,E1 322.110} C_DIS
LIN {X -0.004,Y -228.992,Z 893.770,A 0.000,B 0.000,C 90.000,E1 318.647} C_DIS
LIN {X -0.102,Y -237.949,Z 893.753,A 0.000,B 0.000,C 90.000,E1 315.648} C_DIS
LIN {X -0.141,Y -247.876,Z 893.737,A 0.000,B 0.000,C 90.000,E1 312.690} C_DIS
LIN {X 0.118,Y -258.864,Z 893.721,A 0.000,B 0.000,C 90.000,E1 309.725} C_DIS
LIN {X -0.126,Y -272.417,Z 893.703,A 0.000,B 0.000,C 90.000,E1 306.583} C_DIS
LIN {X -0.021,Y -287.321,Z 893.686,A 0.000,B 0.000,C 90.000,E1 303.452} C_DIS
LIN {X 0.056,Y -303.623,Z 893.669,A 0.000,B 0.000,C 90.000,E1 300.413} C_DIS
LIN {X -0.099,Y -317.577,Z 893.656,A 0.000,B 0.000,C 90.000,E1 298.153} C_DIS
LIN {X 0.019,Y -332.838,Z 893.644,A 0.000,B 0.000,C 90.000,E1 295.899} C_DIS
LIN {X -0.097,Y -352.129,Z 893.630,A 0.000,B 0.000,C 90.000,E1 293.439} C_DIS
LIN {X 0.100,Y -374.734,Z 893.616,A 0.000,B 0.000,C 90.000,E1 290.791} C_DIS
LIN {X 0.201,Y -390.295,Z 893.606,A 0.000,B 0.000,C 90.000,E1 289.087} C_DIS
LIN {X -0.061,Y -405.692,Z 893.597,A 0.000,B 0.000,C 90.000,E1 287.511} C_DIS
LIN {X -0.212,Y -418.242,Z 893.590,A 0.000,B 0.000,C 90.000,E1 286.205} C_DIS
LIN {X 0.130,Y -428.232,Z 893.584,A 0.000,B 0.000,C 90.000,E1 285.079} C_DIS
LIN {X -0.094,Y -440.102,Z 893.576,A 0.000,B 0.000,C 90.000,E1 283.772} C_DIS
LIN {X 0.038,Y -449.031,Z 893.571,A 0.000,B 0.000,C 90.000,E1 282.703} C_DIS
LIN {X 0.050,Y -457.496,Z 893.565,A 0.000,B 0.000,C 90.000,E1 281.658} C_DIS
LIN {X -0.197,Y -465.347,Z 893.559,A 0.000,B 0.000,C 90.000,E1 280.658} C_DIS
LIN {X -0.135,Y -474.440,Z 893.552,A 0.000,B 0.000,C 90.000,E1 279.378} C_DIS
LIN {X -0.155,Y -479.208,Z 893.548,A 0.000,B 0.000,C 90.000,E1 278.624} C_DIS
LIN {X -0.136,Y -483.345,Z 893.544,A 0.000,B 0.000,C 90.000,E1 277.871} C_DIS
LIN {X 0.036,Y -485.701,Z 893.541,A 0.000,B 0.000,C 90.000,E1 277.352} C_DIS
LIN {X 0.227,Y -487.717,Z 893.538,A 0.000,B 0.000,C 90.000,E1 276.834} C_DIS
LIN {X -0.061,Y -489.396,Z 893.535,A 0.000,B 0.000,C 90.000,E1 276.372} C_DIS
LIN {X 0.149,Y -490.712,Z 893.533,A 0.000,B 0.000,C 90.000,E1 275.853} C_DIS
LIN {X -0.121,Y -491.670,Z 893.530,A 0.000,B 0.000,C 90.000,E1 275.391} C_DIS
LIN {X 0.062,Y -492.276,Z 893.527,A 0.000,B 0.000,C 90.000,E1 274.878} C_DIS
LIN {X -0.197,Y -492.466,Z 893.524,A 0.000,B 0.000,C 90.000,E1 274.416} C_DIS
LIN {X 0.037,Y -492.221,Z 893.522,A 0.000,B 0.000,C 90.000,E1 273.898} C_DIS
LIN {X 0.239,Y -491.515,Z 893.519,A 0.000,B 0.000,C 90.000,E1 273.383} C_DIS
LIN {X -0.022,Y -490.372,Z 893.516,A 0.000,B 0.000,C 90.000,E1 272.922} C_DIS
LIN {X 0.177,Y -488.764,Z 893.513,A 0.000,B 0.000,C 90.000,E1 272.407} C_DIS
LIN {X -0.116,Y -486.504,Z 893.511,A 0.000,B 0.000,C 90.000,E1 271.949} C_DIS
LIN {X 0.232,Y -485.251,Z 893.509,A 0.000,B 0.000,C 90.000,E1 271.661} C_DIS
LIN {X -0.081,Y -482.059,Z 893.507,A 0.000,B 0.000,C 90.000,E1 271.203} C_DIS
LIN {X 0.075,Y -478.051,Z 893.504,A 0.000,B 0.000,C 90.000,E1 270.688} C_DIS
LIN {X 0.208,Y -473.082,Z 893.501,A 0.000,B 0.000,C 90.000,E1 270.172} C_DIS
LIN {X 0.051,Y -467.366,Z 893.498,A 0.000,B 0.000,C 90.000,E1 269.714} C_DIS
LIN {X -0.143,Y -461.154,Z 893.496,A 0.000,B 0.000,C 90.000,E1 269.312} C_DIS
LIN {X 0.105,Y -454.538,Z 893.494,A 0.000,B 0.000,C 90.000,E1 268.912} C_DIS
LIN {X -0.145,Y -447.715,Z 893.492,A 0.000,B 0.000,C 90.000,E1 268.625} C_DIS
LIN {X 0.018,Y -440.496,Z 893.491,A 0.000,B 0.000,C 90.000,E1 268.339} C_DIS
LIN {X 0.123,Y -433.001,Z 893.490,A 0.000,B 0.000,C 90.000,E1 268.108} C_DIS
LIN {X 0.131,Y -425.041,Z 893.489,A 0.000,B 0.000,C 90.000,E1 267.936} C_DIS
LIN {X 0.061,Y -415.502,Z 893.488,A 0.000,B 0.000,C 90.000,E1 267.822} C_DIS
LIN {X 0.101,Y -407.184,Z 893.488,A 0.000,B 0.000,C 90.000,E1 267.764} C_DIS
LIN {X 0.022,Y -181.089,Z 893.488,A 0.000,B 0.000,C 90.000,E1 267.764} C_DIS
LIN {X 0.046,Y -180.895,Z 893.473,A 0.000,B 0.000,C 90.000,E1 265.179} C_DIS
